// TIA Portal project "EbAndon v2_0_1" (V15)

(* hardware
DEVICE "S71500/ET200MP station_1"  S7-1500 station
   slot 0: "Rail_0"  Rack  6ES7 590-1***0-0AA0
   slot 1: "PLC_1"  CPU 1515F-2 PN  6ES7 515-2FM01-0AB0  V2.5
      slot 3: "CPU display_1"  6ES7591-1BA00-0AA0
DEVICE "HMI_1"  TP1500 Comfort PRO
   slot 0: "HMI_1"  TP1500 Comfort PRO  6AV2 124-0QC24-1AX0  15.0.0.0
   slot 1: "HMI_RT_1"  TP1500 Comfort PRO  6AV2 124-0QC24-1AX0  15.0.0.0
   slot 5: "HMI_1.IE_CP_1"  PROFINET Interface  15.0.0.0
      slot 1: "PROFINET Interface_1"  PROFINET Interface
         slot 1: "Port_1"  Port
         slot 2: "Port_2"  Port
   slot 6: "HMI_1.IE_CP_2"  PROFINET Interface  15.0.0.0
      slot 1: "PROFINET Interface_GBit"  PROFINET Interface
         slot 1: "Port_1"  Port
   slot 7: "HMI_1.MPI/DP_CP_1"  MPI/DP Interface  15.0.0.0
DEVICE "ET 200SP station_1"  ET 200SP-Station
   slot 0: "Rack_0"  Rack  6ES5 710-8MAx1
   slot 0: "volvo1606et200sp"  IM 155-6 PN ST  6ES7 155-6AU01-0BN0  V4.1
   slot 1: "DQ 8x24VDC/0.5A ST_1"  DQ 8x24VDC/0.5A ST  6ES7 132-6BF01-0BA0  V0.0
      slot 1: "DQ 8x24VDC/0.5A ST_1"  DQ 8x24VDC/0.5A ST
   slot 2: "DQ 8x24VDC/0.5A ST_2"  DQ 8x24VDC/0.5A ST  6ES7 132-6BF01-0BA0  V0.0
      slot 1: "DQ 8x24VDC/0.5A ST_2"  DQ 8x24VDC/0.5A ST
   slot 3: "DQ 8x24VDC/0.5A ST_3"  DQ 8x24VDC/0.5A ST  6ES7 132-6BF01-0BA0  V0.0
      slot 1: "DQ 8x24VDC/0.5A ST_3"  DQ 8x24VDC/0.5A ST
   slot 4: "Server module_1"  Server module  6ES7 193-6PA00-0AA0  V1.1
      slot 1: "Server module_1"  Server module
   slot 127: "BA 2xRJ45"  BA 2xRJ45  6ES7 193-6AR00-0AA0  V0.0
      slot 1: "Port_1"  6ES7 193-6AR00-0AA0  V0.0
      slot 2: "Port_2"  6ES7 193-6AR00-0AA0  V0.0
DEVICE "ET 200SP station_2"  ET 200SP-Station
   slot 0: "Rack_0"  Rack  6ES5 710-8MAx1
   slot 0: "volvo1607et200sp"  IM 155-6 PN ST  6ES7 155-6AU01-0BN0  V4.1
   slot 1: "DQ 8x24VDC/0.5A ST_1"  DQ 8x24VDC/0.5A ST  6ES7 132-6BF01-0BA0  V0.0
      slot 1: "DQ 8x24VDC/0.5A ST_1"  DQ 8x24VDC/0.5A ST
   slot 2: "DQ 8x24VDC/0.5A ST_2"  DQ 8x24VDC/0.5A ST  6ES7 132-6BF01-0BA0  V0.0
      slot 1: "DQ 8x24VDC/0.5A ST_2"  DQ 8x24VDC/0.5A ST
   slot 3: "DQ 8x24VDC/0.5A ST_3"  DQ 8x24VDC/0.5A ST  6ES7 132-6BF01-0BA0  V0.0
      slot 1: "DQ 8x24VDC/0.5A ST_3"  DQ 8x24VDC/0.5A ST
   slot 4: "Server module_1"  Server module  6ES7 193-6PA00-0AA0  V1.1
      slot 1: "Server module_1"  Server module
   slot 127: "BA 2xRJ45"  BA 2xRJ45  6ES7 193-6AR00-0AA0  V0.0
      slot 1: "Port_1"  6ES7 193-6AR00-0AA0  V0.0
      slot 2: "Port_2"  6ES7 193-6AR00-0AA0  V0.0
DEVICE "ET 200SP station_3"  ET 200SP-Station
   slot 0: "Rack_0"  Rack  6ES5 710-8MAx1
   slot 0: "volvo1608et200sp"  IM 155-6 PN ST  6ES7 155-6AU01-0BN0  V4.1
   slot 1: "DQ 8x24VDC/0.5A ST_1"  DQ 8x24VDC/0.5A ST  6ES7 132-6BF01-0BA0  V0.0
      slot 1: "DQ 8x24VDC/0.5A ST_1"  DQ 8x24VDC/0.5A ST
   slot 2: "DQ 8x24VDC/0.5A ST_2"  DQ 8x24VDC/0.5A ST  6ES7 132-6BF01-0BA0  V0.0
      slot 1: "DQ 8x24VDC/0.5A ST_2"  DQ 8x24VDC/0.5A ST
   slot 3: "DQ 8x24VDC/0.5A ST_3"  DQ 8x24VDC/0.5A ST  6ES7 132-6BF01-0BA0  V0.0
      slot 1: "DQ 8x24VDC/0.5A ST_3"  DQ 8x24VDC/0.5A ST
   slot 4: "Server module_1"  Server module  6ES7 193-6PA00-0AA0  V1.1
      slot 1: "Server module_1"  Server module
   slot 127: "BA 2xRJ45"  BA 2xRJ45  6ES7 193-6AR00-0AA0  V0.0
      slot 1: "Port_1"  6ES7 193-6AR00-0AA0  V0.0
      slot 2: "Port_2"  6ES7 193-6AR00-0AA0  V0.0
DEVICE "KP8_1"  SIMATIC Key Panel
   slot 0: "Rack"  Rail  V1.0
   slot 0: "volvo1608kp8"  KP8  6AV3 688-3AY36-0AX0  R01.00.00
DEVICE "KP8_2"  SIMATIC Key Panel
   slot 0: "Rack"  Rail  V1.0
   slot 0: "volvo1607kp8"  KP8  6AV3 688-3AY36-0AX0  R01.00.00
DEVICE "KP8_3"  SIMATIC Key Panel
   slot 0: "Rack"  Rail  V1.0
   slot 0: "volvo1606kp8"  KP8  6AV3 688-3AY36-0AX0  R01.00.00
DEVICE "KP8_4"  SIMATIC Key Panel
   slot 0: "Rack"  Rail  V1.0
   slot 0: "volvo1609kp8"  KP8  6AV3 688-3AY36-0AX0  R01.00.00
DEVICE "ET 200SP station_4"  ET 200SP-Station
   slot 0: "Rack_0"  Rack  6ES5 710-8MAx1
   slot 0: "volvo1609et200sp"  IM 155-6 PN ST  6ES7 155-6AU01-0BN0  V4.1
   slot 1: "DQ 8x24VDC/0.5A ST_1"  DQ 8x24VDC/0.5A ST  6ES7 132-6BF01-0BA0  V0.0
      slot 1: "DQ 8x24VDC/0.5A ST_1"  DQ 8x24VDC/0.5A ST
   slot 2: "DQ 8x24VDC/0.5A ST_2"  DQ 8x24VDC/0.5A ST  6ES7 132-6BF01-0BA0  V0.0
      slot 1: "DQ 8x24VDC/0.5A ST_2"  DQ 8x24VDC/0.5A ST
   slot 3: "DQ 8x24VDC/0.5A ST_3"  DQ 8x24VDC/0.5A ST  6ES7 132-6BF01-0BA0  V0.0
      slot 1: "DQ 8x24VDC/0.5A ST_3"  DQ 8x24VDC/0.5A ST
   slot 4: "Server module_1"  Server module  6ES7 193-6PA00-0AA0  V1.1
      slot 1: "Server module_1"  Server module
   slot 127: "BA 2xRJ45"  BA 2xRJ45  6ES7 193-6AR00-0AA0  V0.0
      slot 1: "Port_1"  6ES7 193-6AR00-0AA0  V0.0
      slot 2: "Port_2"  6ES7 193-6AR00-0AA0  V0.0
DEVICE "ET 200SP station_5"  ET 200SP-Station
   slot 0: "Rack_0"  Rack  6ES5 710-8MAx1
   slot 0: "volvo1610et200sp"  IM 155-6 PN ST  6ES7 155-6AU01-0BN0  V4.1
   slot 1: "DQ 8x24VDC/0.5A ST_1"  DQ 8x24VDC/0.5A ST  6ES7 132-6BF01-0BA0  V0.0
      slot 1: "DQ 8x24VDC/0.5A ST_1"  DQ 8x24VDC/0.5A ST
   slot 2: "DQ 8x24VDC/0.5A ST_2"  DQ 8x24VDC/0.5A ST  6ES7 132-6BF01-0BA0  V0.0
      slot 1: "DQ 8x24VDC/0.5A ST_2"  DQ 8x24VDC/0.5A ST
   slot 3: "DQ 8x24VDC/0.5A ST_3"  DQ 8x24VDC/0.5A ST  6ES7 132-6BF01-0BA0  V0.0
      slot 1: "DQ 8x24VDC/0.5A ST_3"  DQ 8x24VDC/0.5A ST
   slot 4: "Server module_1"  Server module  6ES7 193-6PA00-0AA0  V1.1
      slot 1: "Server module_1"  Server module
   slot 127: "BA 2xRJ45"  BA 2xRJ45  6ES7 193-6AR00-0AA0  V0.0
      slot 1: "Port_1"  6ES7 193-6AR00-0AA0  V0.0
      slot 2: "Port_2"  6ES7 193-6AR00-0AA0  V0.0
DEVICE "KP8_5"  SIMATIC Key Panel
   slot 0: "Rack"  Rail  V1.0
   slot 0: "volvo1610kp8"  KP8  6AV3 688-3AY36-0AX0  R01.00.00
DEVICE "KP8_6"  SIMATIC Key Panel
   slot 0: "Rack"  Rail  V1.0
   slot 0: "volvo1611kp8"  KP8  6AV3 688-3AY36-0AX0  R01.00.00
DEVICE "ET 200SP station_6"  ET 200SP-Station
   slot 0: "Rack_0"  Rack  6ES5 710-8MAx1
   slot 0: "volvo1611et200sp"  IM 155-6 PN ST  6ES7 155-6AU01-0BN0  V4.1
   slot 1: "DQ 8x24VDC/0.5A ST_1"  DQ 8x24VDC/0.5A ST  6ES7 132-6BF01-0BA0  V0.0
      slot 1: "DQ 8x24VDC/0.5A ST_1"  DQ 8x24VDC/0.5A ST
   slot 2: "DQ 8x24VDC/0.5A ST_2"  DQ 8x24VDC/0.5A ST  6ES7 132-6BF01-0BA0  V0.0
      slot 1: "DQ 8x24VDC/0.5A ST_2"  DQ 8x24VDC/0.5A ST
   slot 3: "DQ 8x24VDC/0.5A ST_3"  DQ 8x24VDC/0.5A ST  6ES7 132-6BF01-0BA0  V0.0
      slot 1: "DQ 8x24VDC/0.5A ST_3"  DQ 8x24VDC/0.5A ST
   slot 4: "Server module_1"  Server module  6ES7 193-6PA00-0AA0  V1.1
      slot 1: "Server module_1"  Server module
   slot 127: "BA 2xRJ45"  BA 2xRJ45  6ES7 193-6AR00-0AA0  V0.0
      slot 1: "Port_1"  6ES7 193-6AR00-0AA0  V0.0
      slot 2: "Port_2"  6ES7 193-6AR00-0AA0  V0.0
DEVICE "KP8_7"  SIMATIC Key Panel
   slot 0: "Rack"  Rail  V1.0
   slot 0: "volvo1601kp8"  KP8  6AV3 688-3AY36-0AX0  R01.00.00
DEVICE "ET 200SP station_7"  ET 200SP-Station
   slot 0: "Rack_0"  Rack  6ES5 710-8MAx1
   slot 0: "volvo1601et200sp"  IM 155-6 PN ST  6ES7 155-6AU01-0BN0  V4.1
   slot 1: "DQ 8x24VDC/0.5A ST_1"  DQ 8x24VDC/0.5A ST  6ES7 132-6BF01-0BA0  V0.0
      slot 1: "DQ 8x24VDC/0.5A ST_1"  DQ 8x24VDC/0.5A ST
   slot 2: "DQ 8x24VDC/0.5A ST_2"  DQ 8x24VDC/0.5A ST  6ES7 132-6BF01-0BA0  V0.0
      slot 1: "DQ 8x24VDC/0.5A ST_2"  DQ 8x24VDC/0.5A ST
   slot 3: "DQ 8x24VDC/0.5A ST_3"  DQ 8x24VDC/0.5A ST  6ES7 132-6BF01-0BA0  V0.0
      slot 1: "DQ 8x24VDC/0.5A ST_3"  DQ 8x24VDC/0.5A ST
   slot 4: "Server module_1"  Server module  6ES7 193-6PA00-0AA0  V1.1
      slot 1: "Server module_1"  Server module
   slot 127: "BA 2xRJ45"  BA 2xRJ45  6ES7 193-6AR00-0AA0  V0.0
      slot 1: "Port_1"  6ES7 193-6AR00-0AA0  V0.0
      slot 2: "Port_2"  6ES7 193-6AR00-0AA0  V0.0
DEVICE "ET 200SP station_8"  ET 200SP-Station
   slot 0: "Rack_0"  Rack  6ES5 710-8MAx1
   slot 0: "volvo1602et200sp"  IM 155-6 PN ST  6ES7 155-6AU01-0BN0  V4.1
   slot 1: "DQ 8x24VDC/0.5A ST_1"  DQ 8x24VDC/0.5A ST  6ES7 132-6BF01-0BA0  V0.0
      slot 1: "DQ 8x24VDC/0.5A ST_1"  DQ 8x24VDC/0.5A ST
   slot 2: "DQ 8x24VDC/0.5A ST_2"  DQ 8x24VDC/0.5A ST  6ES7 132-6BF01-0BA0  V0.0
      slot 1: "DQ 8x24VDC/0.5A ST_2"  DQ 8x24VDC/0.5A ST
   slot 3: "DQ 8x24VDC/0.5A ST_3"  DQ 8x24VDC/0.5A ST  6ES7 132-6BF01-0BA0  V0.0
      slot 1: "DQ 8x24VDC/0.5A ST_3"  DQ 8x24VDC/0.5A ST
   slot 4: "Server module_1"  Server module  6ES7 193-6PA00-0AA0  V1.1
      slot 1: "Server module_1"  Server module
   slot 127: "BA 2xRJ45"  BA 2xRJ45  6ES7 193-6AR00-0AA0  V0.0
      slot 1: "Port_1"  6ES7 193-6AR00-0AA0  V0.0
      slot 2: "Port_2"  6ES7 193-6AR00-0AA0  V0.0
DEVICE "KP8_8"  SIMATIC Key Panel
   slot 0: "Rack"  Rail  V1.0
   slot 0: "volvo1602kp8"  KP8  6AV3 688-3AY36-0AX0  R01.00.00
DEVICE "KP8_9"  SIMATIC Key Panel
   slot 0: "Rack"  Rail  V1.0
   slot 0: "volvo1603kp8"  KP8  6AV3 688-3AY36-0AX0  R01.00.00
DEVICE "KP8_10"  SIMATIC Key Panel
   slot 0: "Rack"  Rail  V1.0
   slot 0: "volvo1604kp8"  KP8  6AV3 688-3AY36-0AX0  R01.00.00
DEVICE "KP8_11"  SIMATIC Key Panel
   slot 0: "Rack"  Rail  V1.0
   slot 0: "volvo1605kp8"  KP8  6AV3 688-3AY36-0AX0  R01.00.00
DEVICE "ET 200SP station_9"  ET 200SP-Station
   slot 0: "Rack_0"  Rack  6ES5 710-8MAx1
   slot 0: "volvo1603et200sp"  IM 155-6 PN ST  6ES7 155-6AU01-0BN0  V4.1
   slot 1: "DQ 8x24VDC/0.5A ST_1"  DQ 8x24VDC/0.5A ST  6ES7 132-6BF01-0BA0  V0.0
      slot 1: "DQ 8x24VDC/0.5A ST_1"  DQ 8x24VDC/0.5A ST
   slot 2: "DQ 8x24VDC/0.5A ST_2"  DQ 8x24VDC/0.5A ST  6ES7 132-6BF01-0BA0  V0.0
      slot 1: "DQ 8x24VDC/0.5A ST_2"  DQ 8x24VDC/0.5A ST
   slot 3: "DQ 8x24VDC/0.5A ST_3"  DQ 8x24VDC/0.5A ST  6ES7 132-6BF01-0BA0  V0.0
      slot 1: "DQ 8x24VDC/0.5A ST_3"  DQ 8x24VDC/0.5A ST
   slot 4: "Server module_1"  Server module  6ES7 193-6PA00-0AA0  V1.1
      slot 1: "Server module_1"  Server module
   slot 127: "BA 2xRJ45"  BA 2xRJ45  6ES7 193-6AR00-0AA0  V0.0
      slot 1: "Port_1"  6ES7 193-6AR00-0AA0  V0.0
      slot 2: "Port_2"  6ES7 193-6AR00-0AA0  V0.0
DEVICE "ET 200SP station_10"  ET 200SP-Station
   slot 0: "Rack_0"  Rack  6ES5 710-8MAx1
   slot 0: "volvo1604et200sp"  IM 155-6 PN ST  6ES7 155-6AU01-0BN0  V4.1
   slot 1: "DQ 8x24VDC/0.5A ST_1"  DQ 8x24VDC/0.5A ST  6ES7 132-6BF01-0BA0  V0.0
      slot 1: "DQ 8x24VDC/0.5A ST_1"  DQ 8x24VDC/0.5A ST
   slot 2: "DQ 8x24VDC/0.5A ST_2"  DQ 8x24VDC/0.5A ST  6ES7 132-6BF01-0BA0  V0.0
      slot 1: "DQ 8x24VDC/0.5A ST_2"  DQ 8x24VDC/0.5A ST
   slot 3: "DQ 8x24VDC/0.5A ST_3"  DQ 8x24VDC/0.5A ST  6ES7 132-6BF01-0BA0  V0.0
      slot 1: "DQ 8x24VDC/0.5A ST_3"  DQ 8x24VDC/0.5A ST
   slot 4: "Server module_1"  Server module  6ES7 193-6PA00-0AA0  V1.1
      slot 1: "Server module_1"  Server module
   slot 127: "BA 2xRJ45"  BA 2xRJ45  6ES7 193-6AR00-0AA0  V0.0
      slot 1: "Port_1"  6ES7 193-6AR00-0AA0  V0.0
      slot 2: "Port_2"  6ES7 193-6AR00-0AA0  V0.0
DEVICE "ET 200SP station_11"  ET 200SP-Station
   slot 0: "Rack_0"  Rack  6ES5 710-8MAx1
   slot 0: "volvo1605et200sp"  IM 155-6 PN ST  6ES7 155-6AU01-0BN0  V4.1
   slot 1: "DQ 8x24VDC/0.5A ST_1"  DQ 8x24VDC/0.5A ST  6ES7 132-6BF01-0BA0  V0.0
      slot 1: "DQ 8x24VDC/0.5A ST_1"  DQ 8x24VDC/0.5A ST
   slot 2: "DQ 8x24VDC/0.5A ST_2"  DQ 8x24VDC/0.5A ST  6ES7 132-6BF01-0BA0  V0.0
      slot 1: "DQ 8x24VDC/0.5A ST_2"  DQ 8x24VDC/0.5A ST
   slot 3: "DQ 8x24VDC/0.5A ST_3"  DQ 8x24VDC/0.5A ST  6ES7 132-6BF01-0BA0  V0.0
      slot 1: "DQ 8x24VDC/0.5A ST_3"  DQ 8x24VDC/0.5A ST
   slot 4: "Server module_1"  Server module  6ES7 193-6PA00-0AA0  V1.1
      slot 1: "Server module_1"  Server module
   slot 127: "BA 2xRJ45"  BA 2xRJ45  6ES7 193-6AR00-0AA0  V0.0
      slot 1: "Port_1"  6ES7 193-6AR00-0AA0  V0.0
      slot 2: "Port_2"  6ES7 193-6AR00-0AA0  V0.0
DEVICE "PC-System_1"  SIMATIC PC station
   slot 0: "SIMATIC PC station"  Rail  SIMATIC PC-Station  V1.0
      slot 125: "Stationmanager"  Station_Manager  V6.0.4
   slot 1: "HMI_RT_2"  WinCC RT Advanced  6AV2 104-0xxxx-xxxx  15.0.0.0
      slot 33792: "Host interface"  Host interface
   slot 2: "IE general_1"  IE General  IE_CP  V8.2.0
DEVICE "ET 200SP station_12"  ET 200SP-Station
   slot 0: "Rack_0"  Rack  6ES5 710-8MAx1
   slot 0: "chm01et200sp"  IM 155-6 PN ST  6ES7 155-6AU01-0BN0  V4.1
   slot 1: "DQ 8x24VDC/0.5A ST_1"  DQ 8x24VDC/0.5A ST  6ES7 132-6BF01-0BA0  V0.0
      slot 1: "DQ 8x24VDC/0.5A ST_1"  DQ 8x24VDC/0.5A ST
   slot 2: "DQ 8x24VDC/0.5A ST_2"  DQ 8x24VDC/0.5A ST  6ES7 132-6BF01-0BA0  V0.0
      slot 1: "DQ 8x24VDC/0.5A ST_2"  DQ 8x24VDC/0.5A ST
   slot 3: "DQ 8x24VDC/0.5A ST_3"  DQ 8x24VDC/0.5A ST  6ES7 132-6BF01-0BA0  V0.0
      slot 1: "DQ 8x24VDC/0.5A ST_3"  DQ 8x24VDC/0.5A ST
   slot 4: "Server module_1"  Server module  6ES7 193-6PA00-0AA0  V1.1
      slot 1: "Server module_1"  Server module
   slot 127: "BA 2xRJ45"  BA 2xRJ45  6ES7 193-6AR00-0AA0  V0.0
      slot 1: "Port_1"  6ES7 193-6AR00-0AA0  V0.0
      slot 2: "Port_2"  6ES7 193-6AR00-0AA0  V0.0
DEVICE "KP8_12"  SIMATIC Key Panel
   slot 0: "Rack"  Rail  V1.0
   slot 0: "chm01kp8"  KP8  6AV3 688-3AY36-0AX0  R01.00.00
DEVICE "ET 200SP station_13"  ET 200SP-Station
   slot 0: "Rack_0"  Rack  6ES5 710-8MAx1
   slot 0: "chm02et200sp"  IM 155-6 PN ST  6ES7 155-6AU01-0BN0  V4.1
   slot 1: "DQ 8x24VDC/0.5A ST_1"  DQ 8x24VDC/0.5A ST  6ES7 132-6BF01-0BA0  V0.0
      slot 1: "DQ 8x24VDC/0.5A ST_1"  DQ 8x24VDC/0.5A ST
   slot 2: "DQ 8x24VDC/0.5A ST_2"  DQ 8x24VDC/0.5A ST  6ES7 132-6BF01-0BA0  V0.0
      slot 1: "DQ 8x24VDC/0.5A ST_2"  DQ 8x24VDC/0.5A ST
   slot 3: "DQ 8x24VDC/0.5A ST_3"  DQ 8x24VDC/0.5A ST  6ES7 132-6BF01-0BA0  V0.0
      slot 1: "DQ 8x24VDC/0.5A ST_3"  DQ 8x24VDC/0.5A ST
   slot 4: "Server module_1"  Server module  6ES7 193-6PA00-0AA0  V1.1
      slot 1: "Server module_1"  Server module
   slot 127: "BA 2xRJ45"  BA 2xRJ45  6ES7 193-6AR00-0AA0  V0.0
      slot 1: "Port_1"  6ES7 193-6AR00-0AA0  V0.0
      slot 2: "Port_2"  6ES7 193-6AR00-0AA0  V0.0
DEVICE "KP8_13"  SIMATIC Key Panel
   slot 0: "Rack"  Rail  V1.0
   slot 0: "chm02kp8"  KP8  6AV3 688-3AY36-0AX0  R01.00.00
DEVICE "ET 200SP station_14"  ET 200SP-Station
   slot 0: "Rack_0"  Rack  6ES5 710-8MAx1
   slot 0: "chm03et200sp"  IM 155-6 PN ST  6ES7 155-6AU01-0BN0  V4.1
   slot 1: "DQ 8x24VDC/0.5A ST_1"  DQ 8x24VDC/0.5A ST  6ES7 132-6BF01-0BA0  V0.0
      slot 1: "DQ 8x24VDC/0.5A ST_1"  DQ 8x24VDC/0.5A ST
   slot 2: "DQ 8x24VDC/0.5A ST_2"  DQ 8x24VDC/0.5A ST  6ES7 132-6BF01-0BA0  V0.0
      slot 1: "DQ 8x24VDC/0.5A ST_2"  DQ 8x24VDC/0.5A ST
   slot 3: "DQ 8x24VDC/0.5A ST_3"  DQ 8x24VDC/0.5A ST  6ES7 132-6BF01-0BA0  V0.0
      slot 1: "DQ 8x24VDC/0.5A ST_3"  DQ 8x24VDC/0.5A ST
   slot 4: "Server module_1"  Server module  6ES7 193-6PA00-0AA0  V1.1
      slot 1: "Server module_1"  Server module
   slot 127: "BA 2xRJ45"  BA 2xRJ45  6ES7 193-6AR00-0AA0  V0.0
      slot 1: "Port_1"  6ES7 193-6AR00-0AA0  V0.0
      slot 2: "Port_2"  6ES7 193-6AR00-0AA0  V0.0
DEVICE "KP8_14"  SIMATIC Key Panel
   slot 0: "Rack"  Rail  V1.0
   slot 0: "chm03kp8"  KP8  6AV3 688-3AY36-0AX0  R01.00.00
DEVICE "KP8_15"  SIMATIC Key Panel
   slot 0: "Rack"  Rail  V1.0
   slot 0: "chm04kp8"  KP8  6AV3 688-3AY36-0AX0  R01.00.00
DEVICE "ET 200SP station_15"  ET 200SP-Station
   slot 0: "Rack_0"  Rack  6ES5 710-8MAx1
   slot 0: "chm04et200sp"  IM 155-6 PN ST  6ES7 155-6AU01-0BN0  V4.1
   slot 1: "DQ 8x24VDC/0.5A ST_1"  DQ 8x24VDC/0.5A ST  6ES7 132-6BF01-0BA0  V0.0
      slot 1: "DQ 8x24VDC/0.5A ST_1"  DQ 8x24VDC/0.5A ST
   slot 2: "DQ 8x24VDC/0.5A ST_2"  DQ 8x24VDC/0.5A ST  6ES7 132-6BF01-0BA0  V0.0
      slot 1: "DQ 8x24VDC/0.5A ST_2"  DQ 8x24VDC/0.5A ST
   slot 3: "DQ 8x24VDC/0.5A ST_3"  DQ 8x24VDC/0.5A ST  6ES7 132-6BF01-0BA0  V0.0
      slot 1: "DQ 8x24VDC/0.5A ST_3"  DQ 8x24VDC/0.5A ST
   slot 4: "Server module_1"  Server module  6ES7 193-6PA00-0AA0  V1.1
      slot 1: "Server module_1"  Server module
   slot 127: "BA 2xRJ45"  BA 2xRJ45  6ES7 193-6AR00-0AA0  V0.0
      slot 1: "Port_1"  6ES7 193-6AR00-0AA0  V0.0
      slot 2: "Port_2"  6ES7 193-6AR00-0AA0  V0.0
DEVICE "KP8_16"  SIMATIC Key Panel
   slot 0: "Rack"  Rail  V1.0
   slot 0: "cdo01kp8"  KP8  6AV3 688-3AY36-0AX0  R01.00.00
DEVICE "ET 200SP station_16"  ET 200SP-Station
   slot 0: "Rack_0"  Rack  6ES5 710-8MAx1
   slot 0: "cdo01et200sp"  IM 155-6 PN ST  6ES7 155-6AU01-0BN0  V4.1
   slot 1: "DQ 8x24VDC/0.5A ST_1"  DQ 8x24VDC/0.5A ST  6ES7 132-6BF01-0BA0  V0.0
      slot 1: "DQ 8x24VDC/0.5A ST_1"  DQ 8x24VDC/0.5A ST
   slot 2: "DQ 8x24VDC/0.5A ST_2"  DQ 8x24VDC/0.5A ST  6ES7 132-6BF01-0BA0  V0.0
      slot 1: "DQ 8x24VDC/0.5A ST_2"  DQ 8x24VDC/0.5A ST
   slot 3: "DQ 8x24VDC/0.5A ST_3"  DQ 8x24VDC/0.5A ST  6ES7 132-6BF01-0BA0  V0.0
      slot 1: "DQ 8x24VDC/0.5A ST_3"  DQ 8x24VDC/0.5A ST
   slot 4: "Server module_1"  Server module  6ES7 193-6PA00-0AA0  V1.1
      slot 1: "Server module_1"  Server module
   slot 127: "BA 2xRJ45"  BA 2xRJ45  6ES7 193-6AR00-0AA0  V0.0
      slot 1: "Port_1"  6ES7 193-6AR00-0AA0  V0.0
      slot 2: "Port_2"  6ES7 193-6AR00-0AA0  V0.0
DEVICE "ET 200SP station_17"  ET 200SP-Station
   slot 0: "Rack_0"  Rack  6ES5 710-8MAx1
   slot 0: "cdo02et200sp"  IM 155-6 PN ST  6ES7 155-6AU01-0BN0  V4.1
   slot 1: "DQ 8x24VDC/0.5A ST_1"  DQ 8x24VDC/0.5A ST  6ES7 132-6BF01-0BA0  V0.0
      slot 1: "DQ 8x24VDC/0.5A ST_1"  DQ 8x24VDC/0.5A ST
   slot 2: "DQ 8x24VDC/0.5A ST_2"  DQ 8x24VDC/0.5A ST  6ES7 132-6BF01-0BA0  V0.0
      slot 1: "DQ 8x24VDC/0.5A ST_2"  DQ 8x24VDC/0.5A ST
   slot 3: "DQ 8x24VDC/0.5A ST_3"  DQ 8x24VDC/0.5A ST  6ES7 132-6BF01-0BA0  V0.0
      slot 1: "DQ 8x24VDC/0.5A ST_3"  DQ 8x24VDC/0.5A ST
   slot 4: "Server module_1"  Server module  6ES7 193-6PA00-0AA0  V1.1
      slot 1: "Server module_1"  Server module
   slot 127: "BA 2xRJ45"  BA 2xRJ45  6ES7 193-6AR00-0AA0  V0.0
      slot 1: "Port_1"  6ES7 193-6AR00-0AA0  V0.0
      slot 2: "Port_2"  6ES7 193-6AR00-0AA0  V0.0
DEVICE "KP8_17"  SIMATIC Key Panel
   slot 0: "Rack"  Rail  V1.0
   slot 0: "cdo02kp8"  KP8  6AV3 688-3AY36-0AX0  R01.00.00
DEVICE "KP8_18"  SIMATIC Key Panel
   slot 0: "Rack"  Rail  V1.0
   slot 0: "cdo03kp8"  KP8  6AV3 688-3AY36-0AX0  R01.00.00
DEVICE "ET 200SP station_18"  ET 200SP-Station
   slot 0: "Rack_0"  Rack  6ES5 710-8MAx1
   slot 0: "cdo03et200sp"  IM 155-6 PN ST  6ES7 155-6AU01-0BN0  V4.1
   slot 1: "DQ 8x24VDC/0.5A ST_1"  DQ 8x24VDC/0.5A ST  6ES7 132-6BF01-0BA0  V0.0
      slot 1: "DQ 8x24VDC/0.5A ST_1"  DQ 8x24VDC/0.5A ST
   slot 2: "DQ 8x24VDC/0.5A ST_2"  DQ 8x24VDC/0.5A ST  6ES7 132-6BF01-0BA0  V0.0
      slot 1: "DQ 8x24VDC/0.5A ST_2"  DQ 8x24VDC/0.5A ST
   slot 3: "DQ 8x24VDC/0.5A ST_3"  DQ 8x24VDC/0.5A ST  6ES7 132-6BF01-0BA0  V0.0
      slot 1: "DQ 8x24VDC/0.5A ST_3"  DQ 8x24VDC/0.5A ST
   slot 4: "Server module_1"  Server module  6ES7 193-6PA00-0AA0  V1.1
      slot 1: "Server module_1"  Server module
   slot 127: "BA 2xRJ45"  BA 2xRJ45  6ES7 193-6AR00-0AA0  V0.0
      slot 1: "Port_1"  6ES7 193-6AR00-0AA0  V0.0
      slot 2: "Port_2"  6ES7 193-6AR00-0AA0  V0.0
DEVICE "ET 200SP station_19"  ET 200SP-Station
   slot 0: "Rack_0"  Rack  6ES5 710-8MAx1
   slot 0: "bfl01et200sp"  IM 155-6 PN ST  6ES7 155-6AU01-0BN0  V4.1
   slot 1: "DQ 8x24VDC/0.5A ST_1"  DQ 8x24VDC/0.5A ST  6ES7 132-6BF01-0BA0  V0.0
      slot 1: "DQ 8x24VDC/0.5A ST_1"  DQ 8x24VDC/0.5A ST
   slot 2: "DQ 8x24VDC/0.5A ST_2"  DQ 8x24VDC/0.5A ST  6ES7 132-6BF01-0BA0  V0.0
      slot 1: "DQ 8x24VDC/0.5A ST_2"  DQ 8x24VDC/0.5A ST
   slot 3: "DQ 8x24VDC/0.5A ST_3"  DQ 8x24VDC/0.5A ST  6ES7 132-6BF01-0BA0  V0.0
      slot 1: "DQ 8x24VDC/0.5A ST_3"  DQ 8x24VDC/0.5A ST
   slot 4: "Server module_1"  Server module  6ES7 193-6PA00-0AA0  V1.1
      slot 1: "Server module_1"  Server module
   slot 127: "BA 2xRJ45"  BA 2xRJ45  6ES7 193-6AR00-0AA0  V0.0
      slot 1: "Port_1"  6ES7 193-6AR00-0AA0  V0.0
      slot 2: "Port_2"  6ES7 193-6AR00-0AA0  V0.0
DEVICE "KP8_19"  SIMATIC Key Panel
   slot 0: "Rack"  Rail  V1.0
   slot 0: "bfl01kp8"  KP8  6AV3 688-3AY36-0AX0  R01.00.00
DEVICE "KP8_20"  SIMATIC Key Panel
   slot 0: "Rack"  Rail  V1.0
   slot 0: "bfl02kp8"  KP8  6AV3 688-3AY36-0AX0  R01.00.00
DEVICE "ET 200SP station_20"  ET 200SP-Station
   slot 0: "Rack_0"  Rack  6ES5 710-8MAx1
   slot 0: "bfl02et200sp"  IM 155-6 PN ST  6ES7 155-6AU01-0BN0  V4.1
   slot 1: "DQ 8x24VDC/0.5A ST_1"  DQ 8x24VDC/0.5A ST  6ES7 132-6BF01-0BA0  V0.0
      slot 1: "DQ 8x24VDC/0.5A ST_1"  DQ 8x24VDC/0.5A ST
   slot 2: "DQ 8x24VDC/0.5A ST_2"  DQ 8x24VDC/0.5A ST  6ES7 132-6BF01-0BA0  V0.0
      slot 1: "DQ 8x24VDC/0.5A ST_2"  DQ 8x24VDC/0.5A ST
   slot 3: "DQ 8x24VDC/0.5A ST_3"  DQ 8x24VDC/0.5A ST  6ES7 132-6BF01-0BA0  V0.0
      slot 1: "DQ 8x24VDC/0.5A ST_3"  DQ 8x24VDC/0.5A ST
   slot 4: "Server module_1"  Server module  6ES7 193-6PA00-0AA0  V1.1
      slot 1: "Server module_1"  Server module
   slot 127: "BA 2xRJ45"  BA 2xRJ45  6ES7 193-6AR00-0AA0  V0.0
      slot 1: "Port_1"  6ES7 193-6AR00-0AA0  V0.0
      slot 2: "Port_2"  6ES7 193-6AR00-0AA0  V0.0
DEVICE "ET 200SP station_21"  ET 200SP-Station
   slot 0: "Rack_0"  Rack  6ES5 710-8MAx1
   slot 0: "bfl03et200sp"  IM 155-6 PN ST  6ES7 155-6AU01-0BN0  V4.1
   slot 1: "DQ 8x24VDC/0.5A ST_1"  DQ 8x24VDC/0.5A ST  6ES7 132-6BF01-0BA0  V0.0
      slot 1: "DQ 8x24VDC/0.5A ST_1"  DQ 8x24VDC/0.5A ST
   slot 2: "DQ 8x24VDC/0.5A ST_2"  DQ 8x24VDC/0.5A ST  6ES7 132-6BF01-0BA0  V0.0
      slot 1: "DQ 8x24VDC/0.5A ST_2"  DQ 8x24VDC/0.5A ST
   slot 3: "DQ 8x24VDC/0.5A ST_3"  DQ 8x24VDC/0.5A ST  6ES7 132-6BF01-0BA0  V0.0
      slot 1: "DQ 8x24VDC/0.5A ST_3"  DQ 8x24VDC/0.5A ST
   slot 4: "Server module_1"  Server module  6ES7 193-6PA00-0AA0  V1.1
      slot 1: "Server module_1"  Server module
   slot 127: "BA 2xRJ45"  BA 2xRJ45  6ES7 193-6AR00-0AA0  V0.0
      slot 1: "Port_1"  6ES7 193-6AR00-0AA0  V0.0
      slot 2: "Port_2"  6ES7 193-6AR00-0AA0  V0.0
DEVICE "KP8_21"  SIMATIC Key Panel
   slot 0: "Rack"  Rail  V1.0
   slot 0: "bfl03kp8"  KP8  6AV3 688-3AY36-0AX0  R01.00.00
DEVICE "KP8_22"  SIMATIC Key Panel
   slot 0: "Rack"  Rail  V1.0
   slot 0: "lgs01kp8"  KP8  6AV3 688-3AY36-0AX0  R01.00.00
DEVICE "ET 200SP station_22"  ET 200SP-Station
   slot 0: "Rack_0"  Rack  6ES5 710-8MAx1
   slot 0: "lgs01et200sp"  IM 155-6 PN ST  6ES7 155-6AU01-0BN0  V4.1
   slot 1: "DQ 8x24VDC/0.5A ST_1"  DQ 8x24VDC/0.5A ST  6ES7 132-6BF01-0BA0  V0.0
      slot 1: "DQ 8x24VDC/0.5A ST_1"  DQ 8x24VDC/0.5A ST
   slot 2: "DQ 8x24VDC/0.5A ST_2"  DQ 8x24VDC/0.5A ST  6ES7 132-6BF01-0BA0  V0.0
      slot 1: "DQ 8x24VDC/0.5A ST_2"  DQ 8x24VDC/0.5A ST
   slot 3: "DQ 8x24VDC/0.5A ST_3"  DQ 8x24VDC/0.5A ST  6ES7 132-6BF01-0BA0  V0.0
      slot 1: "DQ 8x24VDC/0.5A ST_3"  DQ 8x24VDC/0.5A ST
   slot 4: "Server module_1"  Server module  6ES7 193-6PA00-0AA0  V1.1
      slot 1: "Server module_1"  Server module
   slot 127: "BA 2xRJ45"  BA 2xRJ45  6ES7 193-6AR00-0AA0  V0.0
      slot 1: "Port_1"  6ES7 193-6AR00-0AA0  V0.0
      slot 2: "Port_2"  6ES7 193-6AR00-0AA0  V0.0
DEVICE "ET 200SP station_23"  ET 200SP-Station
   slot 0: "Rack_0"  Rack  6ES5 710-8MAx1
   slot 0: "lgs02et200sp"  IM 155-6 PN ST  6ES7 155-6AU01-0BN0  V4.1
   slot 1: "DQ 8x24VDC/0.5A ST_1"  DQ 8x24VDC/0.5A ST  6ES7 132-6BF01-0BA0  V0.0
      slot 1: "DQ 8x24VDC/0.5A ST_1"  DQ 8x24VDC/0.5A ST
   slot 2: "DQ 8x24VDC/0.5A ST_2"  DQ 8x24VDC/0.5A ST  6ES7 132-6BF01-0BA0  V0.0
      slot 1: "DQ 8x24VDC/0.5A ST_2"  DQ 8x24VDC/0.5A ST
   slot 3: "DQ 8x24VDC/0.5A ST_3"  DQ 8x24VDC/0.5A ST  6ES7 132-6BF01-0BA0  V0.0
      slot 1: "DQ 8x24VDC/0.5A ST_3"  DQ 8x24VDC/0.5A ST
   slot 4: "Server module_1"  Server module  6ES7 193-6PA00-0AA0  V1.1
      slot 1: "Server module_1"  Server module
   slot 127: "BA 2xRJ45"  BA 2xRJ45  6ES7 193-6AR00-0AA0  V0.0
      slot 1: "Port_1"  6ES7 193-6AR00-0AA0  V0.0
      slot 2: "Port_2"  6ES7 193-6AR00-0AA0  V0.0
DEVICE "KP8_23"  SIMATIC Key Panel
   slot 0: "Rack"  Rail  V1.0
   slot 0: "lgs02kp8"  KP8  6AV3 688-3AY36-0AX0  R01.00.00
DEVICE "KP8_24"  SIMATIC Key Panel
   slot 0: "Rack"  Rail  V1.0
   slot 0: "chm05kp8"  KP8  6AV3 688-3AY36-0AX0  R01.00.00
DEVICE "ET 200SP station_24"  ET 200SP-Station
   slot 0: "Rack_0"  Rack  6ES5 710-8MAx1
   slot 0: "chm05et200sp"  IM 155-6 PN ST  6ES7 155-6AU01-0BN0  V4.1
   slot 1: "DQ 8x24VDC/0.5A ST_1"  DQ 8x24VDC/0.5A ST  6ES7 132-6BF01-0BA0  V0.0
      slot 1: "DQ 8x24VDC/0.5A ST_1"  DQ 8x24VDC/0.5A ST
   slot 2: "DQ 8x24VDC/0.5A ST_2"  DQ 8x24VDC/0.5A ST  6ES7 132-6BF01-0BA0  V0.0
      slot 1: "DQ 8x24VDC/0.5A ST_2"  DQ 8x24VDC/0.5A ST
   slot 3: "DQ 8x24VDC/0.5A ST_3"  DQ 8x24VDC/0.5A ST  6ES7 132-6BF01-0BA0  V0.0
      slot 1: "DQ 8x24VDC/0.5A ST_3"  DQ 8x24VDC/0.5A ST
   slot 4: "Server module_1"  Server module  6ES7 193-6PA00-0AA0  V1.1
      slot 1: "Server module_1"  Server module
   slot 127: "BA 2xRJ45"  BA 2xRJ45  6ES7 193-6AR00-0AA0  V0.0
      slot 1: "Port_1"  6ES7 193-6AR00-0AA0  V0.0
      slot 2: "Port_2"  6ES7 193-6AR00-0AA0  V0.0
*)

// ===== PLC "PLC_1"  CPU 1515F-2 PN =====

VAR_GLOBAL   // PLC tag table "Default tag table"
   "System_Byte" AT %MB1 : Byte;
   "FirstScan" AT %M1.0 : Bool;
   "DiagStatusUpdate" AT %M1.1 : Bool;
   "AlwaysTRUE" AT %M1.2 : Bool;
   "AlwaysFALSE" AT %M1.3 : Bool;
   "Clock_Byte" AT %MB0 : Byte;
   "Clock_10Hz" AT %M0.0 : Bool;
   "Clock_5Hz" AT %M0.1 : Bool;
   "Clock_2.5Hz" AT %M0.2 : Bool;
   "Clock_2Hz" AT %M0.3 : Bool;
   "Clock_1.25Hz" AT %M0.4 : Bool;
   "Clock_1Hz" AT %M0.5 : Bool;
   "Clock_0.625Hz" AT %M0.6 : Bool;
   "Clock_0.5Hz" AT %M0.7 : Bool;
   "Temp Reset" AT %M2.0 : Bool;
   "clearPartData" AT %M100.0 : Bool;
   "setDefaultPresets" AT %M100.1 : Bool;
   "hardInitReq" AT %M100.2 : Bool;
END_VAR

VAR_GLOBAL   // PLC tag table "VOLVO 16 01"
   "VOLVO 16 01 IO" AT %QD100 : DWord;
   "VOLVO 16 01 KP8 In" AT %ID0 : DWord;
   "VOLVO 16 01 KP8 Out" AT %QD0 : DWord;
END_VAR

VAR_GLOBAL   // PLC tag table "VOLVO 16 02"
   "VOLVO 16 02 IO" AT %QD104 : DWord;
   "VOLVO 16 02 KP8 In" AT %ID4 : DWord;
   "VOLVO 16 02 KP8 Out" AT %QD4 : DWord;
END_VAR

VAR_GLOBAL   // PLC tag table "VOLVO 16 03"
   "VOLVO 16 03 IO" AT %QD108 : DWord;
   "VOLVO 16 03 KP8 In" AT %ID8 : DWord;
   "VOLVO 16 03 KP8 Out" AT %QD8 : DWord;
END_VAR

VAR_GLOBAL   // PLC tag table "VOLVO 16 04"
   "VOLVO 16 04 IO" AT %QD112 : DWord;
   "VOLVO 16 04 KP8 In" AT %ID12 : DWord;
   "VOLVO 16 04 KP8 Out" AT %QD12 : DWord;
END_VAR

VAR_GLOBAL   // PLC tag table "VOLVO 16 05"
   "VOLVO 16 05 IO" AT %QD116 : DWord;
   "VOLVO 16 05 KP8 In" AT %ID16 : DWord;
   "VOLVO 16 05 KP8 Out" AT %QD16 : DWord;
END_VAR

VAR_GLOBAL   // PLC tag table "VOLVO 16 06"
   "VOLVO 16 06 IO" AT %QD120 : DWord;
   "VOLVO 16 06 KP8 In" AT %ID20 : DWord;
   "VOLVO 16 06 KP8 Out" AT %QD20 : DWord;
END_VAR

VAR_GLOBAL   // PLC tag table "VOLVO 16 07"
   "VOLVO 16 07 IO" AT %QD124 : DWord;
   "VOLVO 16 07 KP8 In" AT %ID24 : DWord;
   "VOLVO 16 07 KP8 Out" AT %QD24 : DWord;
END_VAR

VAR_GLOBAL   // PLC tag table "VOLVO 16 08"
   "VOLVO 16 08 IO" AT %QD128 : DWord;
   "VOLVO 16 08 KP8 In" AT %ID28 : DWord;
   "VOLVO 16 08 KP8 Out" AT %QD28 : DWord;
END_VAR

VAR_GLOBAL   // PLC tag table "VOLVO 16 09"
   "VOLVO 16 09 IO" AT %QD132 : DWord;
   "VOLVO 16 09 KP8 In" AT %ID32 : DWord;
   "VOLVO 16 09 KP8 Out" AT %QD32 : DWord;
END_VAR

VAR_GLOBAL   // PLC tag table "VOLVO 16 10"
   "VOLVO 16 10 IO" AT %QD136 : DWord;
   "VOLVO 16 10 KP8 In" AT %ID36 : DWord;
   "VOLVO 16 10 KP8 Out" AT %QD36 : DWord;
END_VAR

VAR_GLOBAL   // PLC tag table "VOLVO 16 11"
   "VOLVO 16 11 IO" AT %QD140 : DWord;
   "VOLVO 16 11 KP8 In" AT %ID40 : DWord;
   "VOLVO 16 11 KP8 Out" AT %QD40 : DWord;
END_VAR

VAR_GLOBAL   // PLC tag table "CHM 02"
   "CHM 02 KP8 In" AT %ID44 : DWord;
   "CHM 02 KP8 Out" AT %QD44 : DWord;
   "CHM 02 IO" AT %QD144 : DWord;
END_VAR

VAR_GLOBAL   // PLC tag table "CHM 03"
   "CHM 03 IO" AT %QD148 : DWord;
   "CHM 03 KP8 In" AT %ID48 : DWord;
   "CHM 03 KP8 Out" AT %QD48 : DWord;
END_VAR

VAR_GLOBAL   // PLC tag table "CHM 04"
   "CHM 04 IO" AT %QD152 : DWord;
   "CHM 04 KP8 In" AT %ID52 : DWord;
   "CHM 04 KP8 Out" AT %QD52 : DWord;
END_VAR

VAR_GLOBAL   // PLC tag table "CHM 05"
   "CHM 05 IO" AT %QD156 : DWord;
   "CHM 05 KP8 In" AT %ID56 : DWord;
   "CHM 05 KP8 Out" AT %QD56 : DWord;
END_VAR

VAR_GLOBAL   // PLC tag table "CDO 01"
   "CDO 01 IO" AT %QD160 : DWord;
   "CDO 01 KP8 In" AT %ID60 : DWord;
   "CDO 01 KP8 Out" AT %QD60 : DWord;
END_VAR

VAR_GLOBAL   // PLC tag table "CDO 02"
   "CDO 02 IO" AT %QD164 : DWord;
   "CDO 02 KP8 In" AT %ID64 : DWord;
   "CDO 02 KP8 Out" AT %QD64 : DWord;
END_VAR

VAR_GLOBAL   // PLC tag table "CDO 03"
   "CDO 03 IO" AT %QD168 : DWord;
   "CDO 03 KP8 In" AT %ID68 : DWord;
   "CDO 03 KP8 Out" AT %QD68 : DWord;
END_VAR

VAR_GLOBAL   // PLC tag table "BFL 01"
   "BFL 01 IO" AT %QD172 : DWord;
   "BFL 01 KP8 In" AT %ID72 : DWord;
   "BFL 01 KP8 Out" AT %QD72 : DWord;
END_VAR

VAR_GLOBAL   // PLC tag table "BFL 02"
   "BFL 02 IO" AT %QD176 : DWord;
   "BFL 02 KP8 In" AT %ID76 : DWord;
   "BFL 02 KP8 Out" AT %QD76 : DWord;
END_VAR

VAR_GLOBAL   // PLC tag table "BFL 03"
   "BFL 03 IO" AT %QD180 : DWord;
   "BFL 03 KP8 In" AT %ID80 : DWord;
   "BFL 03 KP8 Out" AT %QD80 : DWord;
END_VAR

VAR_GLOBAL   // PLC tag table "LGS 01"
   "LGS 01 IO" AT %QD184 : DWord;
   "LGS 01 KP8 In" AT %ID84 : DWord;
   "LGS 01 KP8 Out" AT %QD84 : DWord;
END_VAR

VAR_GLOBAL   // PLC tag table "LGS 02"
   "LGS 02 IO" AT %QD188 : DWord;
   "LGS 02 KP8 In" AT %ID88 : DWord;
   "LGS 02 KP8 Out" AT %QD88 : DWord;
END_VAR

VAR_GLOBAL   // PLC tag table "CHM 01"
   "CHM 01 IO" AT %QD192 : DWord;
   "CHM 01 KP8 In" AT %ID92 : DWord;
   "CHM 01 KP8 Out" AT %QD92 : DWord;
END_VAR

TYPE "Stations"
   STRUCT
      current : Array[0..23] of "Station";
      old : Array[0..23] of "Station";
   END_STRUCT;
END_TYPE

TYPE "Part Call Screen"
   STRUCT
      current : Array[0..11] of "Table Row";
   END_STRUCT;
END_TYPE

TYPE "Settings Screen"
   STRUCT
      current : "Settings";
   END_STRUCT;
END_TYPE

TYPE "Barcode Screen"
   STRUCT
      partNumber : WString[40];
      barcode : String;
      orderCancelled : Bool;
      ordered : Bool;
   END_STRUCT;
END_TYPE

TYPE "Table Row"
   STRUCT
      address : UInt;
      ordered : Bool;
      pbSelection : Struct
         actuate : Bool;
         animate : USInt;
      END_STRUCT;
      rtBackground : Struct
         animate : USInt;
      END_STRUCT;
      tfDropZone : Struct
         animate : USInt;
         value : WString[20];
      END_STRUCT;
      tfLine : Struct
         animate : USInt;
         value : WString[20];
      END_STRUCT;
      tfPartNumber : Struct
         animate : USInt;
         value : WString[40];
      END_STRUCT;
      tfTime : Struct
         animate : UInt;
         value : WString[20];
      END_STRUCT;
   END_STRUCT;
END_TYPE

TYPE "Runtime Data"
   STRUCT
      asReal : Real;
      elapsed : LReal;
      mem : LReal;
   END_STRUCT;
END_TYPE

TYPE "KP8 Button Config"
   STRUCT
      activate : Array[0..7] of Bool;
      colorOn1 : Array[0..7] of String[10];
      colorOn2 : Array[0..7] of String[10];
      colorOff : Array[0..7] of String[10];
      flash : Array[0..7] of Bool;
      group : Array[0..7] of Int;
      mode : Array[0..7] of Bool;
   END_STRUCT;
END_TYPE

TYPE "Constants"
   STRUCT
      buttonCount : Int := 6;   // max buttons per station
      hmiRowCount : Int := 11;   // number of rows displayed on hmi
      stationCount : Int := 24;   // total number of stations
      hmiSelStnCount : Int := 12;   // labels for settings screen
      defaultAlotted : Real := 1800.0;
      defaultCritical : Real := 300.0;
      partReqRows : Int := 200;
      ledRowCount : Int := 11;
      colorLib : "Color Library";
   END_STRUCT;
END_TYPE

TYPE "Part Request Data"
   STRUCT
      row : Array[0..199] of "Table Row";
   END_STRUCT;
END_TYPE

TYPE "Station"
   STRUCT
      animations : Array[0..7] of Int;
      btnStates : Array[0..7] of Bool;
      dropZone : USInt;
      elapsedTime : Struct
         partReq : Array[0..7] of Real;
         resetReq : Real;
      END_STRUCT;
      kp8Config : "KP8 Button Config";
      kp8In : Byte;
      kp8Out : DWord;
      init : Struct
         hard : Bool;
         soft : Bool;
      END_STRUCT;
      line : WString[20];
      partNumbers : Array[0..7] of WString[40];
      partOrdered : Array[0..7] of Bool;
      presetTime : Struct
         allotted : Array[0..7] of Real;
         critical : Array[0..7] of Real;
      END_STRUCT;
      stackLightOut : DWord;
      settings : Struct
         selected : Bool;
         btnSelection : Array[0..7] of Bool;
      END_STRUCT;
   END_STRUCT;
END_TYPE

TYPE "Settings"
   STRUCT
      alotted : Struct
         assign : "PB Data: Text Label";
         ioField : "IO Field Data: Timers";
      END_STRUCT;
      critical : Struct
         assign : "PB Data: Text Label";
         ioField : "IO Field Data: Timers";
      END_STRUCT;
      kp8 : Struct
         selectButtons : "PB Data: Text Label";
         btnSelState : Array[0..7] of Bool;
         buttons : Array[0..7] of "PB Data: Text Label";
         selBtnNumber : Int;
         selCount : Int;
      END_STRUCT;
      stations : Struct
         selectAll : "PB Data: Text Label";
         nextGroup : "PB Data: Graphic/Text List";
         prevGroup : "PB Data: Graphic/Text List";
         selectBtns : Array[0..11] of "PB Data: Text Label";
         selCount : Int;
      END_STRUCT;
      partNumber : Struct
         assign : "PB Data: Text Label";
         ioField : "IO Field Data: Part Number";
      END_STRUCT;
      viewingStation : Struct
         btns : Array[0..5] of "Station Assignment: Button Details";
         dzData : "Drop Zone Data";
         lineData : "Line Label Data";
         next : "PB Data: Graphic/Text List";
         previous : "PB Data: Graphic/Text List";
         "name" : WString[20];
      END_STRUCT;
   END_STRUCT;
END_TYPE

TYPE "PB Data: Graphic/Text List"
   STRUCT
      actuate : Bool;
      animate : USInt;
      listSelect : UInt;
   END_STRUCT;
END_TYPE

TYPE "LED Sign Data"
   STRUCT
      row : Array[0..11] of "Table Row";
   END_STRUCT;
END_TYPE

TYPE "PB Data: Text Label"
   STRUCT
      actuate : Bool;
      animate : USInt;
      label : WString[20];
   END_STRUCT;
END_TYPE

TYPE "Color Library"
   STRUCT
      BkBk : USInt := 0;
      BgWh : USInt := 1;
      FgWh : USInt := 2;
      FlWh : USInt := 3;
      BgGray : USInt := 4;
      FgGray : USInt := 5;
      FlGray : USInt := 6;
      BgLRd : USInt := 7;
      FgLRd : USInt := 8;
      FlLRd : USInt := 9;
      BgDRd : USInt := 10;
      FgDRd : USInt := 11;
      FlDrd : USInt := 12;
      BgLYe : USInt := 13;
      FgLYe : USInt := 14;
      FlLYe : USInt := 15;
      BgDYe : USInt := 16;
      FgDYe : USInt := 17;
      FlDYe : USInt := 18;
      BgLGr : USInt := 19;
      FgLGr : USInt := 20;
      FlLGr : USInt := 21;
      BgDGr : USInt := 22;
      FgDGr : USInt := 23;
      FlDGr : USInt := 24;
      BgLTe : USInt := 25;
      FgLTe : USInt := 26;
      FlLTe : USInt := 27;
      BgDTe : USInt := 28;
      FgDTe : USInt := 29;
      FlDTe : USInt := 30;
      BgLBl : USInt := 31;
      FgLBl : USInt := 32;
      FlLBl : USInt := 33;
      BgDBl : USInt := 34;
      FgDBl : USInt := 35;
      FlDBl : USInt := 36;
      BgLPu : USInt := 37;
      FgLPu : USInt := 38;
      FlLPu : USInt := 39;
      BgDPu : USInt := 40;
      FgDPu : USInt := 41;
      FlDPu : USInt := 42;
      disabled : USInt := 254;
      invisible : USInt := 255;
   END_STRUCT;
END_TYPE

TYPE "Station Assignment: Button Details"
   STRUCT
      alloted : Struct
         animate : USInt;
         value : WString[10];
      END_STRUCT;
      critical : Struct
         animate : USInt;
         value : WString[10];
      END_STRUCT;
      label : Struct
         animate : USInt;
         value : WString[2];
      END_STRUCT;
      partNumber : Struct
         animate : USInt;
         value : WString[40];
      END_STRUCT;
      select : Struct
         actuate : Bool;
         animate : USInt;
      END_STRUCT;
   END_STRUCT;
END_TYPE

TYPE "IO Field Data: Part Number"
   STRUCT
      animate : USInt;
      inputFinished : Bool;
      value : WString[40];
   END_STRUCT;
END_TYPE

TYPE "Line Label Data"
   STRUCT
      animate : Struct
         bg : USInt;
         ioField : USInt;
      END_STRUCT;
      inputFinished : Bool;
      value : WString[10];
   END_STRUCT;
END_TYPE

TYPE "Drop Zone Data"
   STRUCT
      animate : Struct
         bg : USInt;
         ioField : USInt;
      END_STRUCT;
      inputFinished : Bool;
      value : WString[10];
   END_STRUCT;
END_TYPE

TYPE "IO Field Data: Timers"
   STRUCT
      animate : USInt;
      inputFinished : Bool;
      value : WString[5];
   END_STRUCT;
END_TYPE

DATA_BLOCK "EMP IDB"   // DB1
{ S7_Optimized_Access := 'TRUE' }
VERSION : 0.1
// stored: InstanceOfName EMP
"EMP"
BEGIN
   constants.buttonCount := 8;
   stations.current[0].presetTime.allotted[7] := 1800.0;
   stations.current[0].presetTime.allotted[3] := 1800.0;
   stations.current[0].presetTime.critical[7] := 300.0;
   stations.current[0].presetTime.critical[3] := 300.0;
   stations.current[0].partNumbers[7] := WSTRING#'16.32.112.500.100A';
   stations.current[0].partNumbers[6] := WSTRING#'';
   stations.current[0].partNumbers[5] := WSTRING#'';
   stations.current[0].partNumbers[3] := WSTRING#'16.32.112.500.220A';
   stations.current[0].partNumbers[2] := WSTRING#'';
   stations.current[0].partNumbers[1] := WSTRING#'';
   stations.current[0].line := WSTRING#'VOLVO 16';
   stations.current[1].line := WSTRING#'VOLVO 16';
   stations.current[2].line := WSTRING#'VOLVO 16';
   stations.current[0].dropZone := 1;
   stations.current[1].dropZone := 2;
   stations.current[2].dropZone := 3;
   stations.current[3].dropZone := 4;
   stations.current[3].line := WSTRING#'VOLVO 16';
   stations.current[4].dropZone := 5;
   stations.current[4].line := WSTRING#'VOLVO 16';
   stations.current[5].line := WSTRING#'VOLVO 16';
   stations.current[5].dropZone := 6;
   stations.current[6].dropZone := 7;
   stations.current[6].line := WSTRING#'VOLVO 16';
   stations.current[7].dropZone := 8;
   stations.current[7].line := WSTRING#'VOLVO 16';
   stations.current[8].dropZone := 9;
   stations.current[8].line := WSTRING#'VOLVO 16';
   stations.current[9].dropZone := 10;
   stations.current[9].line := WSTRING#'VOLVO 16';
   stations.current[10].dropZone := 11;
   stations.current[10].line := WSTRING#'VOLVO 16';
   stations.current[11].line := WSTRING#'CHM';
   stations.current[11].dropZone := 1;
   stations.current[12].line := WSTRING#'CHM';
   stations.current[12].dropZone := 2;
   stations.current[13].line := WSTRING#'CHM';
   stations.current[13].dropZone := 3;
   stations.current[14].dropZone := 4;
   stations.current[14].line := WSTRING#'CHM';
   stations.current[15].line := WSTRING#'CHM';
   stations.current[15].dropZone := 5;
   stations.current[16].dropZone := 1;
   stations.current[16].line := WSTRING#'CDO';
   stations.current[17].dropZone := 2;
   stations.current[17].line := WSTRING#'CDO';
   stations.current[18].line := WSTRING#'CDO';
   stations.current[18].dropZone := 3;
   stations.current[19].dropZone := 1;
   stations.current[19].line := WSTRING#'BFL';
   stations.current[20].dropZone := 2;
   stations.current[20].line := WSTRING#'BFL';
   stations.current[21].line := WSTRING#'BFL';
   stations.current[21].dropZone := 3;
   stations.current[22].dropZone := 1;
   stations.current[22].line := WSTRING#'LGS';
   stations.current[22].partNumbers[7] := WSTRING#'16.08.216.161.020A';
   stations.current[21].partNumbers[5] := WSTRING#'';
   stations.current[21].partNumbers[6] := WSTRING#'';
   stations.current[21].partNumbers[7] := WSTRING#'16.08.208.011.010G';
   stations.current[18].partNumbers[3] := WSTRING#'16.08.216.911.040B$L16.08.216.200.050A';
   stations.current[18].partNumbers[4] := WSTRING#'';
   stations.current[18].partNumbers[5] := WSTRING#'';
   stations.current[18].partNumbers[6] := WSTRING#'16.08.216.181.020A$L16.08.208.331.000F';
   stations.current[18].partNumbers[7] := WSTRING#'16.08.216.951.010A';
   stations.current[19].partNumbers[7] := WSTRING#'16.08.211.511.020F';
   stations.current[11].partNumbers[0] := WSTRING#'';
   stations.current[11].partNumbers[1] := WSTRING#'';
   stations.current[11].partNumbers[2] := WSTRING#'';
   stations.current[11].partNumbers[3] := WSTRING#'16.08.216.515.008C';
   stations.current[11].partNumbers[4] := WSTRING#'';
   stations.current[11].partNumbers[5] := WSTRING#'';
   stations.current[11].partNumbers[6] := WSTRING#'';
   stations.current[11].partNumbers[7] := WSTRING#'16.08.208.131.010L';
   stations.current[13].partNumbers[0] := WSTRING#'';
   stations.current[13].partNumbers[1] := WSTRING#'';
   stations.current[13].partNumbers[2] := WSTRING#'16.08.216.251.000B';
   stations.current[13].partNumbers[3] := WSTRING#'16.08.216.911.000G';
   stations.current[13].partNumbers[4] := WSTRING#'';
   stations.current[13].partNumbers[5] := WSTRING#'';
   stations.current[13].partNumbers[6] := WSTRING#'16.08.216.911.000H';
   stations.current[13].partNumbers[7] := WSTRING#'16.08.216.911.000C';
   stations.current[14].partNumbers[0] := WSTRING#'';
   stations.current[14].partNumbers[1] := WSTRING#'';
   stations.current[14].partNumbers[2] := WSTRING#'16.08.216.181.100A';
   stations.current[14].partNumbers[3] := WSTRING#'16.08.216.910.020B';
   stations.current[14].partNumbers[4] := WSTRING#'';
   stations.current[14].partNumbers[5] := WSTRING#'16.08.216.181.090A';
   stations.current[14].partNumbers[6] := WSTRING#'16.08.216.722.001A';
   stations.current[14].partNumbers[7] := WSTRING#'16.08.216.181.010B';
   stations.current[18].partNumbers[0] := WSTRING#'';
   stations.current[18].partNumbers[1] := WSTRING#'';
   stations.current[18].partNumbers[2] := WSTRING#'';
   stations.current[12].partNumbers[0] := WSTRING#'';
   stations.current[12].partNumbers[1] := WSTRING#'16.08.216.526.009A';
   stations.current[12].partNumbers[2] := WSTRING#'16.08.216.871.010C';
   stations.current[12].partNumbers[3] := WSTRING#'16.08.216.141.010C';
   stations.current[12].partNumbers[4] := WSTRING#'';
   stations.current[12].partNumbers[5] := WSTRING#'16.08.216.526.002C';
   stations.current[12].partNumbers[6] := WSTRING#'16.08.215.871.010C';
   stations.current[12].partNumbers[7] := WSTRING#'16.08.215.141.010C';
   stations.current[17].partNumbers[0] := WSTRING#'';
   stations.current[17].partNumbers[1] := WSTRING#'';
   stations.current[17].partNumbers[2] := WSTRING#'16.08.216.501.010A';
   stations.current[17].partNumbers[3] := WSTRING#'16.08.208.691.010D';
   stations.current[17].partNumbers[4] := WSTRING#'';
   stations.current[17].partNumbers[5] := WSTRING#'';
   stations.current[17].partNumbers[6] := WSTRING#'16.08.216.790.001A';
   stations.current[17].partNumbers[7] := WSTRING#'16.08.208.531.020L';
   stations.current[15].partNumbers[0] := WSTRING#'';
   stations.current[15].partNumbers[1] := WSTRING#'';
   stations.current[15].partNumbers[2] := WSTRING#'16.08.216.511.000C';
   stations.current[15].partNumbers[3] := WSTRING#'16.08.208.501.000B';
   stations.current[15].partNumbers[4] := WSTRING#'';
   stations.current[15].partNumbers[5] := WSTRING#'16.08.216.551.000B';
   stations.current[15].partNumbers[6] := WSTRING#'16.08.216.231.000B';
   stations.current[15].partNumbers[7] := WSTRING#'16.08.216.501.000C';
   stations.current[16].partNumbers[0] := WSTRING#'';
   stations.current[16].partNumbers[1] := WSTRING#'';
   stations.current[16].partNumbers[2] := WSTRING#'';
   stations.current[16].partNumbers[3] := WSTRING#'16.08.216.912.060B$L16.08.216.202.080A';
   stations.current[16].partNumbers[4] := WSTRING#'';
   stations.current[16].partNumbers[5] := WSTRING#'';
   stations.current[16].partNumbers[6] := WSTRING#'16.08.216.911.030B';
   stations.current[16].partNumbers[7] := WSTRING#'16.08.216.912.050A';
   stations.current[21].partNumbers[0] := WSTRING#'';
   stations.current[21].partNumbers[1] := WSTRING#'';
   stations.current[21].partNumbers[2] := WSTRING#'';
   stations.current[21].partNumbers[3] := WSTRING#'';
   stations.current[21].partNumbers[4] := WSTRING#'';
   stations.current[20].partNumbers[0] := WSTRING#'';
   stations.current[20].partNumbers[1] := WSTRING#'';
   stations.current[20].partNumbers[2] := WSTRING#'';
   stations.current[20].partNumbers[3] := WSTRING#'';
   stations.current[20].partNumbers[4] := WSTRING#'';
   stations.current[20].partNumbers[5] := WSTRING#'';
   stations.current[20].partNumbers[6] := WSTRING#'';
   stations.current[20].partNumbers[7] := WSTRING#'PEANUTS';
   stations.current[8].partNumbers[0] := WSTRING#'';
   stations.current[8].partNumbers[1] := WSTRING#'';
   stations.current[8].partNumbers[2] := WSTRING#'';
   stations.current[8].partNumbers[3] := WSTRING#'16.32.112.580.020A';
   stations.current[8].partNumbers[4] := WSTRING#'';
   stations.current[8].partNumbers[5] := WSTRING#'';
   stations.current[8].partNumbers[6] := WSTRING#'16.32.112.500.300E';
   stations.current[8].partNumbers[7] := WSTRING#'16.32.112.520.300E';
   stations.current[9].partNumbers[0] := WSTRING#'';
   stations.current[9].partNumbers[1] := WSTRING#'';
   stations.current[9].partNumbers[2] := WSTRING#'';
   stations.current[9].partNumbers[3] := WSTRING#'16.32.112.594.000C';
   stations.current[9].partNumbers[4] := WSTRING#'';
   stations.current[9].partNumbers[5] := WSTRING#'';
   stations.current[9].partNumbers[6] := WSTRING#'';
   stations.current[9].partNumbers[7] := WSTRING#'16.32.112.584.000C';
   stations.current[10].partNumbers[0] := WSTRING#'';
   stations.current[10].partNumbers[1] := WSTRING#'';
   stations.current[10].partNumbers[2] := WSTRING#'';
   stations.current[10].partNumbers[3] := WSTRING#'16.32.112.500.150B';
   stations.current[10].partNumbers[4] := WSTRING#'';
   stations.current[10].partNumbers[5] := WSTRING#'';
   stations.current[10].partNumbers[6] := WSTRING#'16.32.806.502.080A';
   stations.current[10].partNumbers[7] := WSTRING#'16.32.112.500.160A';
   stations.current[0].partNumbers[0] := WSTRING#'';
   stations.current[0].partNumbers[4] := WSTRING#'';
   stations.current[1].partNumbers[0] := WSTRING#'';
   stations.current[1].partNumbers[1] := WSTRING#'';
   stations.current[1].partNumbers[2] := WSTRING#'16.32.112.509.070A';
   stations.current[1].partNumbers[3] := WSTRING#'16.32.112.704.000C';
   stations.current[1].partNumbers[4] := WSTRING#'';
   stations.current[1].partNumbers[5] := WSTRING#'';
   stations.current[1].partNumbers[6] := WSTRING#'16.32.112.504.060A';
   stations.current[1].partNumbers[7] := WSTRING#'16.32.112.500.060D';
   stations.current[2].partNumbers[0] := WSTRING#'';
   stations.current[2].partNumbers[1] := WSTRING#'16.32.112.509.050E';
   stations.current[2].partNumbers[2] := WSTRING#'16.32.112.504.070G';
   stations.current[2].partNumbers[3] := WSTRING#'16.32.112.851.001A';
   stations.current[2].partNumbers[4] := WSTRING#'';
   stations.current[2].partNumbers[5] := WSTRING#'16.32.112.509.080F';
   stations.current[2].partNumbers[6] := WSTRING#'16.32.112.870.000C';
   stations.current[2].partNumbers[7] := WSTRING#'16.32.112.851.000A';
   stations.current[3].partNumbers[0] := WSTRING#'';
   stations.current[3].partNumbers[1] := WSTRING#'16.32.112.522.130A';
   stations.current[3].partNumbers[2] := WSTRING#'16.32.112.522.050A';
   stations.current[3].partNumbers[3] := WSTRING#'16.32.112.521.020B';
   stations.current[3].partNumbers[4] := WSTRING#'';
   stations.current[3].partNumbers[5] := WSTRING#'16.32.112.522.040D';
   stations.current[3].partNumbers[6] := WSTRING#'16.32.112.521.010B';
   stations.current[3].partNumbers[7] := WSTRING#'16.32.112.521.030A';
   stations.current[4].partNumbers[0] := WSTRING#'';
   stations.current[4].partNumbers[1] := WSTRING#'';
   stations.current[4].partNumbers[2] := WSTRING#'';
   stations.current[4].partNumbers[3] := WSTRING#'';
   stations.current[4].partNumbers[4] := WSTRING#'';
   stations.current[4].partNumbers[5] := WSTRING#'';
   stations.current[4].partNumbers[6] := WSTRING#'';
   stations.current[4].partNumbers[7] := WSTRING#'16.32.112.529.020B';
   stations.current[5].partNumbers[0] := WSTRING#'';
   stations.current[5].partNumbers[1] := WSTRING#'16.32.112.529.010A';
   stations.current[5].partNumbers[2] := WSTRING#'16.32.112.529.030A';
   stations.current[5].partNumbers[3] := WSTRING#'16.32.112.502.060B';
   stations.current[5].partNumbers[4] := WSTRING#'';
   stations.current[5].partNumbers[5] := WSTRING#'16.32.112.529.050D';
   stations.current[5].partNumbers[6] := WSTRING#'16.32.112.502.070E';
   stations.current[5].partNumbers[7] := WSTRING#'16.32.112.502.050B';
   stations.current[6].partNumbers[0] := WSTRING#'';
   stations.current[6].partNumbers[1] := WSTRING#'16.32.112.621.020A';
   stations.current[6].partNumbers[2] := WSTRING#'16.32.112.621.010A';
   stations.current[6].partNumbers[3] := WSTRING#'16.32.112.751.000D';
   stations.current[6].partNumbers[4] := WSTRING#'';
   stations.current[6].partNumbers[5] := WSTRING#'16.32.112.751.001C';
   stations.current[6].partNumbers[6] := WSTRING#'16.32.112.601.040A';
   stations.current[6].partNumbers[7] := WSTRING#'16.32.112.601.030A';
   stations.current[7].partNumbers[0] := WSTRING#'';
   stations.current[7].partNumbers[1] := WSTRING#'';
   stations.current[7].partNumbers[2] := WSTRING#'';
   stations.current[7].partNumbers[3] := WSTRING#'16.32.112.500.520B';
   stations.current[7].partNumbers[4] := WSTRING#'';
   stations.current[7].partNumbers[5] := WSTRING#'';
   stations.current[7].partNumbers[6] := WSTRING#'16.32.112.500.090B';
   stations.current[7].partNumbers[7] := WSTRING#'16.32.112.500.120A';
   stations.current[23].line := WSTRING#'LGS';
   stations.current[23].dropZone := 2;
   stations.current[23].partNumbers[0] := WSTRING#'';
   stations.current[23].partNumbers[1] := WSTRING#'';
   stations.current[23].partNumbers[2] := WSTRING#'';
   stations.current[23].partNumbers[3] := WSTRING#'';
   stations.current[23].partNumbers[4] := WSTRING#'';
   stations.current[23].partNumbers[5] := WSTRING#'';
   stations.current[23].partNumbers[6] := WSTRING#'';
   stations.current[23].partNumbers[7] := WSTRING#'16.08.208.021.020C';
   stations.current[22].partNumbers[0] := WSTRING#'';
   stations.current[22].partNumbers[1] := WSTRING#'';
   stations.current[22].partNumbers[2] := WSTRING#'';
   stations.current[22].partNumbers[3] := WSTRING#'16.08.208.161.020F';
   stations.current[22].partNumbers[4] := WSTRING#'';
   stations.current[22].partNumbers[5] := WSTRING#'';
   stations.current[22].partNumbers[6] := WSTRING#'OP60 - STAMPINGS';
   stations.current[19].partNumbers[0] := WSTRING#'';
   stations.current[19].partNumbers[1] := WSTRING#'';
   stations.current[19].partNumbers[2] := WSTRING#'16.08.216.831.020A';
   stations.current[19].partNumbers[3] := WSTRING#'16.08.208.151.010F';
   stations.current[19].partNumbers[4] := WSTRING#'';
   stations.current[19].partNumbers[5] := WSTRING#'16.08.217.411.080A';
   stations.current[19].partNumbers[6] := WSTRING#'16.08.216.151.010B';
   constants.hmiRowCount := 12;
END_DATA_BLOCK

DATA_BLOCK "HMI"   // DB2
{ S7_Optimized_Access := 'TRUE' }
VERSION : 0.1
   VAR
      partCall : "Part Call Screen";
      screenNumber : Int;
      settings : "Settings Screen";
      barcode : "Barcode Screen";
   END_VAR
BEGIN
   settings.current.kp8.buttons[1].label := WSTRING#'6';
   settings.current.kp8.buttons[2].label := WSTRING#'4';
   settings.current.kp8.buttons[3].label := WSTRING#'2';
   settings.current.kp8.buttons[5].label := WSTRING#'5';
   settings.current.kp8.buttons[6].label := WSTRING#'3';
   settings.current.kp8.buttons[7].label := WSTRING#'1';
END_DATA_BLOCK

DATA_BLOCK "Parts"   // DB3
{ S7_Optimized_Access := 'TRUE' }
VERSION : 0.1
   VAR
      pRow : Int;
   END_VAR
   VAR RETAIN
      requests : "Part Request Data";
   END_VAR
BEGIN
END_DATA_BLOCK

DATA_BLOCK "LED Sign"   // DB4
{ S7_Optimized_Access := 'TRUE' }
VERSION : 0.1
   VAR
      request : "LED Sign Data";
   END_VAR
BEGIN
END_DATA_BLOCK

FUNCTION_BLOCK "EMP"   // FB1, LAD
{ S7_Optimized_Access := 'TRUE' }
VERSION : 0.1
   VAR RETAIN
      constants : "Constants";
   END_VAR
   VAR
      instBaseAnimations : "Base Animations";
      instHMIAnimations : "Format Part Call Requests";
      instInitialize : "Initialize";
      instKP8ButtonActivation : "KP8 Button Activation";
      instKP8ExpandedAnimations : "KP8 Expanded Animations";
      instPartTimers : "Part Timers";
      instRecordPartRequest : "Record Part Request";
      instRemovePartRequest : "Remove Part Request";
      instResetInitRequest : "Reset Init Requests";
      instStackLightAnimations : "Stack Light Animations";
      "KP8 Drivers" : Array[0..#stationCount] of "KP8 Driver";
   END_VAR
   VAR RETAIN
      stations : "Stations";
   END_VAR
   VAR
      instHMIBarcode : "HMI Barcod Screen";
      instCollapseTable : "Collapse Table";
      instPopulateHMI : "HMI Populate Part Call";
      instHMISettings : "HMI Settings Screen";
      instClearReqData : "Clear Part Requests";
      instDefaultTmrPrst : "Load Default Timer Presets";
      instPopulateLED : "LED Populate Sign";
   END_VAR
   VAR_TEMP
      i : Int;
      stnCount : Int;
   END_VAR
   VAR CONSTANT
      stationCount : Int := 24;
   END_VAR
BEGIN

REGION Network 1: PHYSICAL TO GLOBAL
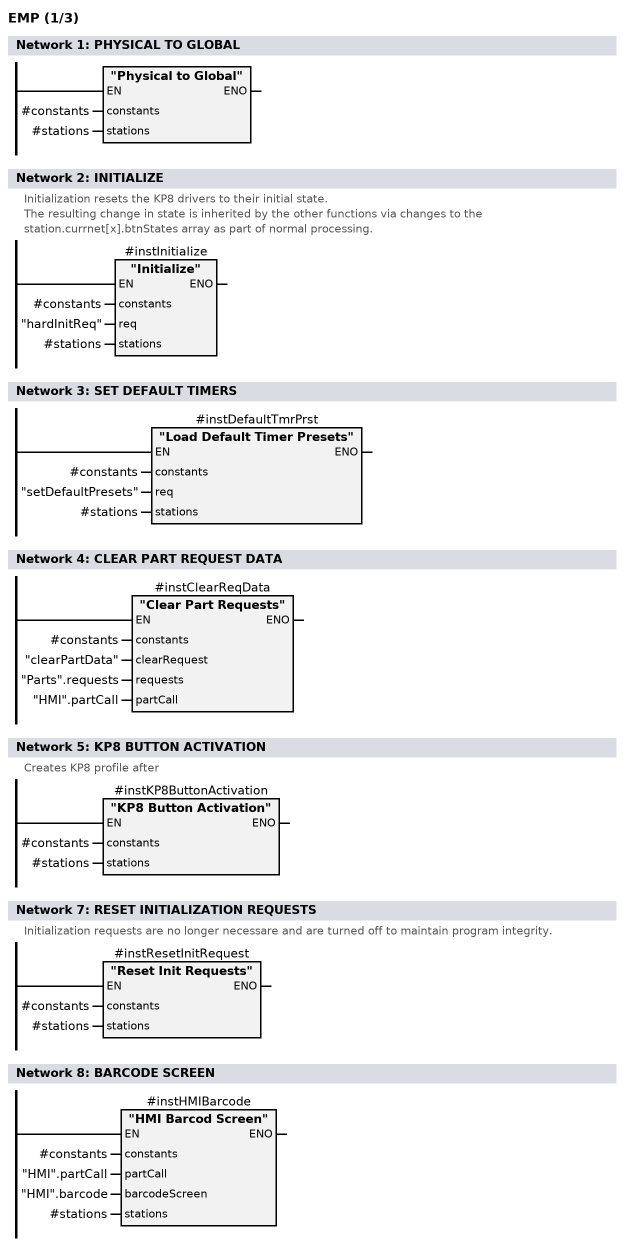
   RUNG wire#powerrail
      "Physical to Global"(constants := #constants, stations := #stations)
   END_RUNG
   // the same network as SCL:
   "Physical to Global"(constants := #constants, stations := #stations);
END_REGION

REGION Network 2: INITIALIZE
   // Initialization resets the KP8 drivers to their initial state.
   // The resulting change in state is inherited by the other functions via changes to the
   // station.currnet[x].btnStates array as part of normal processing.
   RUNG wire#powerrail
      #instInitialize(constants := #constants, req := "hardInitReq", stations := #stations)
   END_RUNG
   // the same network as SCL:
   #instInitialize(constants := #constants, req := "hardInitReq", stations := #stations);   // "Initialize"
END_REGION

REGION Network 3: SET DEFAULT TIMERS
   RUNG wire#powerrail
      #instDefaultTmrPrst(constants := #constants, req := "setDefaultPresets", stations := #stations)
   END_RUNG
   // the same network as SCL:
   #instDefaultTmrPrst(constants := #constants, req := "setDefaultPresets", stations := #stations);   // "Load Default Timer Presets"
END_REGION

REGION Network 4: CLEAR PART REQUEST DATA
   RUNG wire#powerrail
      #instClearReqData(constants := #constants, clearRequest := "clearPartData", requests := "Parts".requests, partCall := "HMI".partCall)
   END_RUNG
   // the same network as SCL:
   #instClearReqData(constants := #constants,   // "Clear Part Requests"
                     clearRequest := "clearPartData",
                     requests := "Parts".requests,
                     partCall := "HMI".partCall);
END_REGION

REGION Network 5: KP8 BUTTON ACTIVATION
   // Creates KP8 profile after
   RUNG wire#powerrail
      #instKP8ButtonActivation(constants := #constants, stations := #stations)
   END_RUNG
   // the same network as SCL:
   #instKP8ButtonActivation(constants := #constants, stations := #stations);   // "KP8 Button Activation"
END_REGION

REGION Network 6 (SCL): KP8 DRIVER CALLS
   REGION "LOOP THROUGH STATIONS"
       #stnCount := #constants.stationCount - 1;
       FOR #i := 0 TO #stnCount DO
           #"KP8 Drivers"[#i](btnIn := #stations.current[#i].kp8In,
                              hardInit := #stations.current[#i].init.hard,
                              softInit := #stations.current[#i].init.soft,
                              btn0Activate := #stations.current[#i].kp8Config.activate[0],
                              btn0Mode := #stations.current[#i].kp8Config.mode[0],
                              btn0Group := #stations.current[#i].kp8Config.group[0],
                              btn0Flash := #stations.current[#i].kp8Config.flash[0],
                              btn0ColorOn1 := #stations.current[#i].kp8Config.colorOn1[0],
                              btn0ColorOn2 := #stations.current[#i].kp8Config.colorOn2[0],
                              btn0ColorOff := #stations.current[#i].kp8Config.colorOff[0],
                              btn1Activate := #stations.current[#i].kp8Config.activate[1],
                              btn1Mode := #stations.current[#i].kp8Config.mode[1],
                              btn1Group := #stations.current[#i].kp8Config.group[1],
                              btn1Flash := #stations.current[#i].kp8Config.flash[1],
                              btn1ColorOn1 := #stations.current[#i].kp8Config.colorOn1[1],
                              btn1ColorOn2 := #stations.current[#i].kp8Config.colorOn2[1],
                              btn1ColorOff := #stations.current[#i].kp8Config.colorOff[1],
                              btn2Activate := #stations.current[#i].kp8Config.activate[2],
                              btn2Mode := #stations.current[#i].kp8Config.mode[2],
                              btn2Group := #stations.current[#i].kp8Config.group[2],
                              btn2Flash := #stations.current[#i].kp8Config.flash[2],
                              btn2ColorOn1 := #stations.current[#i].kp8Config.colorOn1[2],
                              btn2ColorOn2 := #stations.current[#i].kp8Config.colorOn2[2],
                              btn2ColorOff := #stations.current[#i].kp8Config.colorOff[2],
                              btn3Activate := #stations.current[#i].kp8Config.activate[3],
                              btn3Mode := #stations.current[#i].kp8Config.mode[3],
                              btn3Group := #stations.current[#i].kp8Config.group[3],
                              btn3Flash := #stations.current[#i].kp8Config.flash[3],
                              btn3ColorOn1 := #stations.current[#i].kp8Config.colorOn1[3],
                              btn3ColorOn2 := #stations.current[#i].kp8Config.colorOn2[3],
                              btn3ColorOff := #stations.current[#i].kp8Config.colorOff[3],
                              btn4Activate := #stations.current[#i].kp8Config.activate[4],
                              btn4Mode := #stations.current[#i].kp8Config.mode[4],
                              btn4Group := #stations.current[#i].kp8Config.group[4],
                              btn4Flash := #stations.current[#i].kp8Config.flash[4],
                              btn4ColorOn1 := #stations.current[#i].kp8Config.colorOn1[4],
                              btn4ColorOn2 := #stations.current[#i].kp8Config.colorOn2[4],
                              btn4ColorOff := #stations.current[#i].kp8Config.colorOff[4],
                              btn5Activate := #stations.current[#i].kp8Config.activate[5],
                              btn5Mode := #stations.current[#i].kp8Config.mode[5],
                              btn5Group := #stations.current[#i].kp8Config.group[5],
                              btn5Flash := #stations.current[#i].kp8Config.flash[5],
                              btn5ColorOn1 := #stations.current[#i].kp8Config.colorOn1[5],
                              btn5ColorOn2 := #stations.current[#i].kp8Config.colorOn2[5],
                              btn5ColorOff := #stations.current[#i].kp8Config.colorOff[5],
                              btn6Activate := #stations.current[#i].kp8Config.activate[6],
                              btn6Mode := #stations.current[#i].kp8Config.mode[6],
                              btn6Group := #stations.current[#i].kp8Config.group[6],
                              btn6Flash := #stations.current[#i].kp8Config.flash[6],
                              btn6ColorOn1 := #stations.current[#i].kp8Config.colorOn1[6],
                              btn6ColorOn2 := #stations.current[#i].kp8Config.colorOn2[6],
                              btn6ColorOff := #stations.current[#i].kp8Config.colorOff[6],
                              btn7Activate := #stations.current[#i].kp8Config.activate[7],
                              btn7Mode := #stations.current[#i].kp8Config.mode[7],
                              btn7Group := #stations.current[#i].kp8Config.group[7],
                              btn7Flash := #stations.current[#i].kp8Config.flash[7],
                              btn7ColorOn1 := #stations.current[#i].kp8Config.colorOn1[7],
                              btn7ColorOn2 := #stations.current[#i].kp8Config.colorOn2[7],
                              btn7ColorOff := #stations.current[#i].kp8Config.colorOff[7],
                              btnStatesOut => #stations.current[#i].btnStates,
                              btnColorsOut => #stations.current[#i].kp8Out);
       END_FOR;
   END_REGION
END_REGION

REGION Network 7: RESET INITIALIZATION REQUESTS
   // Initialization requests are no longer necessare and are turned off to maintain program integrity.
   RUNG wire#powerrail
      #instResetInitRequest(constants := #constants, stations := #stations)
   END_RUNG
   // the same network as SCL:
   #instResetInitRequest(constants := #constants, stations := #stations);   // "Reset Init Requests"
END_REGION

REGION Network 8: BARCODE SCREEN
   RUNG wire#powerrail
      #instHMIBarcode(constants := #constants, partCall := "HMI".partCall, barcodeScreen := "HMI".barcode, stations := #stations)
   END_RUNG
   // the same network as SCL:
   #instHMIBarcode(constants := #constants,   // "HMI Barcod Screen"
                   partCall := "HMI".partCall,
                   barcodeScreen := "HMI".barcode,
                   stations := #stations);
END_REGION

REGION Network 9: PART TIMERS
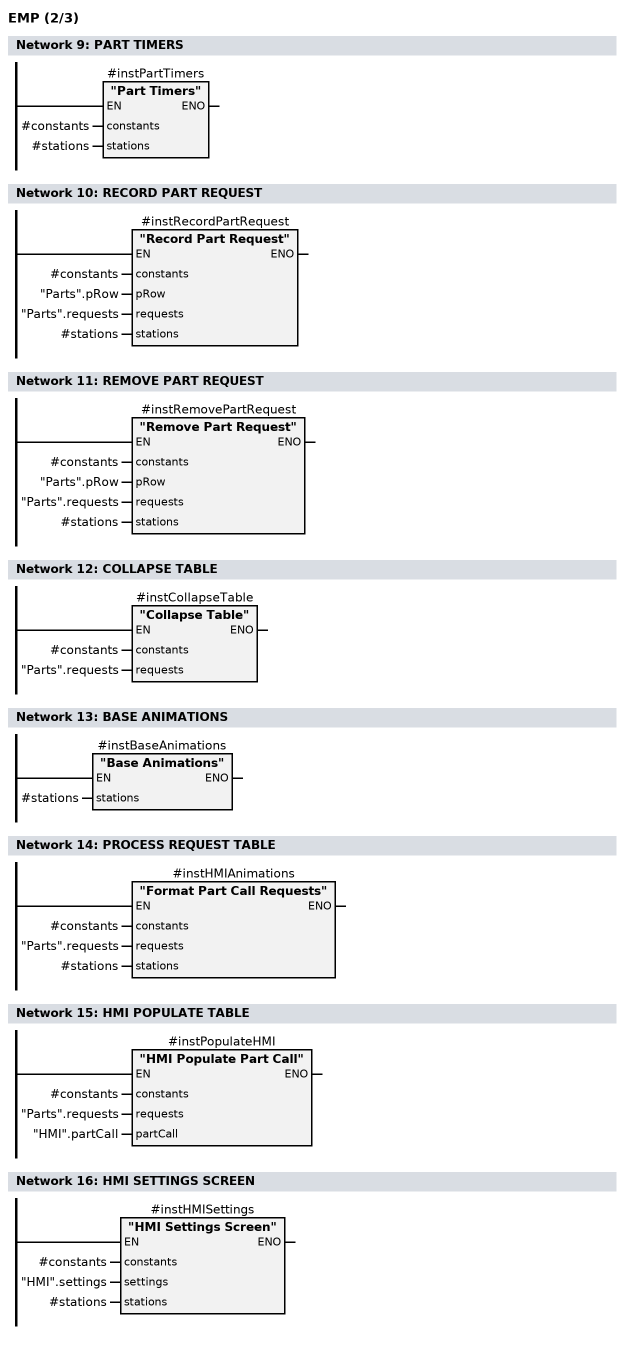
   RUNG wire#powerrail
      #instPartTimers(constants := #constants, stations := #stations)
   END_RUNG
   // the same network as SCL:
   #instPartTimers(constants := #constants, stations := #stations);   // "Part Timers"
END_REGION

REGION Network 10: RECORD PART REQUEST
   RUNG wire#powerrail
      #instRecordPartRequest(constants := #constants, pRow := "Parts".pRow, requests := "Parts".requests, stations := #stations)
   END_RUNG
   // the same network as SCL:
   #instRecordPartRequest(constants := #constants,   // "Record Part Request"
                          pRow := "Parts".pRow,
                          requests := "Parts".requests,
                          stations := #stations);
END_REGION

REGION Network 11: REMOVE PART REQUEST
   RUNG wire#powerrail
      #instRemovePartRequest(constants := #constants, pRow := "Parts".pRow, requests := "Parts".requests, stations := #stations)
   END_RUNG
   // the same network as SCL:
   #instRemovePartRequest(constants := #constants,   // "Remove Part Request"
                          pRow := "Parts".pRow,
                          requests := "Parts".requests,
                          stations := #stations);
END_REGION

REGION Network 12: COLLAPSE TABLE
   RUNG wire#powerrail
      #instCollapseTable(constants := #constants, requests := "Parts".requests)
   END_RUNG
   // the same network as SCL:
   #instCollapseTable(constants := #constants, requests := "Parts".requests);   // "Collapse Table"
END_REGION

REGION Network 13: BASE ANIMATIONS
   RUNG wire#powerrail
      #instBaseAnimations(stations := #stations)
   END_RUNG
   // the same network as SCL:
   #instBaseAnimations(stations := #stations);   // "Base Animations"
END_REGION

REGION Network 14: PROCESS REQUEST TABLE
   RUNG wire#powerrail
      #instHMIAnimations(constants := #constants, requests := "Parts".requests, stations := #stations)
   END_RUNG
   // the same network as SCL:
   #instHMIAnimations(constants := #constants, requests := "Parts".requests, stations := #stations);   // "Format Part Call Requests"
END_REGION

REGION Network 15: HMI POPULATE TABLE
   RUNG wire#powerrail
      #instPopulateHMI(constants := #constants, requests := "Parts".requests, partCall := "HMI".partCall)
   END_RUNG
   // the same network as SCL:
   #instPopulateHMI(constants := #constants, requests := "Parts".requests, partCall := "HMI".partCall);   // "HMI Populate Part Call"
END_REGION

REGION Network 16: HMI SETTINGS SCREEN
   RUNG wire#powerrail
      #instHMISettings(constants := #constants, settings := "HMI".settings, stations := #stations)
   END_RUNG
   // the same network as SCL:
   #instHMISettings(constants := #constants, settings := "HMI".settings, stations := #stations);   // "HMI Settings Screen"
END_REGION

REGION Network 17: LED POPULATE SIGN
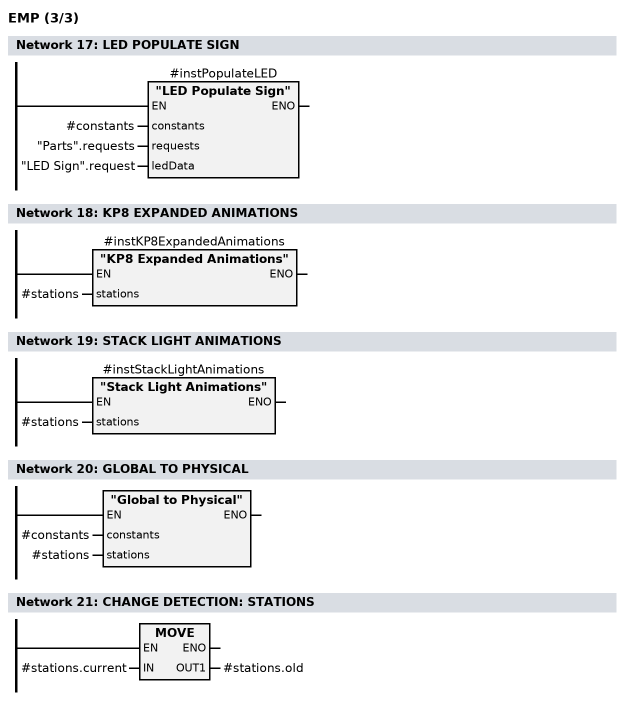
   RUNG wire#powerrail
      #instPopulateLED(constants := #constants, requests := "Parts".requests, ledData := "LED Sign".request)
   END_RUNG
   // the same network as SCL:
   #instPopulateLED(constants := #constants, requests := "Parts".requests, ledData := "LED Sign".request);   // "LED Populate Sign"
END_REGION

REGION Network 18: KP8 EXPANDED ANIMATIONS
   RUNG wire#powerrail
      #instKP8ExpandedAnimations(stations := #stations)
   END_RUNG
   // the same network as SCL:
   #instKP8ExpandedAnimations(stations := #stations);   // "KP8 Expanded Animations"
END_REGION

REGION Network 19: STACK LIGHT ANIMATIONS
   RUNG wire#powerrail
      #instStackLightAnimations(stations := #stations)
   END_RUNG
   // the same network as SCL:
   #instStackLightAnimations(stations := #stations);   // "Stack Light Animations"
END_REGION

REGION Network 20: GLOBAL TO PHYSICAL
   RUNG wire#powerrail
      "Global to Physical"(constants := #constants, stations := #stations)
   END_RUNG
   // the same network as SCL:
   "Global to Physical"(constants := #constants, stations := #stations);
END_REGION

REGION Network 21: CHANGE DETECTION: STATIONS
   RUNG wire#powerrail
      Move(in := #stations.current, out1 => #stations.old)
   END_RUNG
   // the same network as SCL:
   #stations.old := #stations.current;
END_REGION
END_FUNCTION_BLOCK

FUNCTION_BLOCK "Code 128"   // FB2, SCL
{ S7_Optimized_Access := 'TRUE' }
VERSION : 0.1
   VAR_INPUT
      partNumber : String;
   END_VAR
   VAR_OUTPUT
      barcode : String;
   END_VAR
   VAR
      charsIn : Array[0..255] of Byte;
      charsOut : Array[0..255] of Byte;
      cnt : UInt;
      intVals : Array[0..255] of Int;
      sum : Int;
      checkSum : Int;
   END_VAR
   VAR_TEMP
      pn : String;
      i : Int;
   END_VAR
   VAR CONSTANT
      startChar : Char := 'Ì';
      stopChar : Char := 'Î';
   END_VAR
   // intVals[0] := 104;
BEGIN
   #pn := #partNumber;

   FOR #i := 0 TO 255 DO
       #charsIn[#i] := 16#00;
       #charsOut[#i] := 16#00;
       #intVals[#i] := 0;
   END_FOR;

   Strg_TO_Chars(Strg:=#pn,
                 pChars:=0,
                 Cnt=>#cnt,
                 Chars:=#charsIn);


   #sum := 104;
   FOR #i := 0 TO UINT_TO_INT(#cnt - 1) DO
       #intVals[#i] := CHAR_TO_INT(#charsIn[#i]) - 32;
       #intVals[#i] := #intVals[#i] * (#i + 1);
       #sum := #sum + #intVals[#i];
   END_FOR;
   #checkSum := (#sum MOD 103) + 32;
   IF #checkSum >= 127 THEN
       #checkSum := #checkSum + 68;
   END_IF;

   #charsOut[0] := #startChar;
   FOR #i := 1 TO UINT_TO_INT(#cnt) DO
       #charsOut[#i] := #charsIn[#i - 1];
   END_FOR;
   #charsOut[#cnt + 1] := INT_TO_BYTE(#checkSum);
   #charsOut[#cnt + 2] := INT_TO_BYTE(#stopChar);

   Chars_TO_Strg(Chars := #charsOut,
                 pChars := 0,
                 Cnt := #cnt + 3,
                 Strg => #barcode);
END_FUNCTION_BLOCK

FUNCTION_BLOCK "HMI Barcod Screen"   // FB3, SCL
{ S7_Optimized_Access := 'TRUE' }
VERSION : 0.1
   VAR_INPUT
      constants : "Constants";
   END_VAR
   VAR_IN_OUT
      partCall : "Part Call Screen";
      barcodeScreen : "Barcode Screen";
      stations : "Stations";
   END_VAR
   VAR
      address : UInt;
      button : UInt;
      instCode128 : "Code 128";
      codeOut : String;
      pnOut : WString[40];
      station : UInt;
      oldSelectedRow : Int;
   END_VAR
   VAR_TEMP
      orderCancelled : Int;
      processedPN : String[40];
      selectedPN : String[40];
      userOrdered : Bool;
      selectedRow : Int;
   END_VAR
   VAR CONSTANT
      maxRows : Int := 199;
   END_VAR
BEGIN
   REGION "GET USER ROW SELECTION"
       #selectedRow := "Get Part Call Row Number"(constants := #constants,
                                                  partCall := #partCall);
   END_REGION

   REGION "ON SELECTION OF A PART CALL ROW
       IF #selectedRow <> 0 THEN
           IF #selectedRow <> #oldSelectedRow THEN

               REGION "GET BUTTON AND STATION NUMBERS"
                   #address := #partCall.current[#selectedRow - 1].address;
                   "Address to Station and Button"(address := #address,
                                                   station => #station,
                                                   button => #button);
               END_REGION

               REGION "CONVERT STRING TO BARCODE"

                   REGION "COPY TO LOCALS"
                       #selectedPN := WSTRING_TO_STRING(#partCall.current[#selectedRow - 1].tfPartNumber.value);
                   END_REGION

                   REGION "CONVERT TO BARCODE"
                       #instCode128(partNumber := #processedPN,
                                    barcode => #codeOut);
                   END_REGION

                   REGION "OUTPUT FOR HMI SCREEN"
                       #barcodeScreen.partNumber := STRING_TO_WSTRING(#processedPN);
                       #barcodeScreen.barcode := #codeOut;
                   END_REGION

               END_REGION

           END_IF;
       END_IF;
   END_REGION

   REGION "PASS USER ORDERED"
       // get input
       #userOrdered := #barcodeScreen.ordered;
       // put into station
       #stations.current[#station].partOrdered[#button] := #userOrdered;
   END_REGION


   #oldSelectedRow := #selectedRow;
END_FUNCTION_BLOCK

FUNCTION_BLOCK "Initialize"   // FB4, SCL
{ S7_Optimized_Access := 'TRUE' }
VERSION : 0.1
   VAR_INPUT
      constants : "Constants";
      req : Bool;
   END_VAR
   VAR_IN_OUT
      stations : "Stations";
   END_VAR
   VAR
      rtElapsed : Real;
      rt : Struct
         elapsed : LReal;
         mem : LReal;
      END_STRUCT;
   END_VAR
   VAR_TEMP
      i : Int;
      reset : Struct
         req : Bool;
         elapsed : Real;
      END_STRUCT;
      stnCount : Int;
      init : Bool;
   END_VAR
   VAR CONSTANT
      resetLimit : Real := 1.25;
   END_VAR
BEGIN
   REGION "GET STATION COUNT"
       #stnCount := #constants.stationCount - 1;
   END_REGION

   REGION "FIRST SCAN OR REQUEST"
       IF "FirstScan" OR #req THEN
           // initialize all stations on plc first scan
           FOR #i := 0 TO #stnCount DO
               #stations.current[#i].init.hard := TRUE;
           END_FOR;
       END_IF;
   END_REGION

   REGION "RUNTIME CALL"
       // get elapsed time
       #rt.elapsed := RUNTIME(#rt.mem);
       // convert to real data type
       #rtElapsed := LREAL_TO_REAL(#rt.elapsed);
   END_REGION

   REGION "BUTTON 0 BASED RESET TIMERS"
       FOR #i := 0 TO #stnCount DO

           REGION "PRE-CONDITION"
               // init off by default
               #init := FALSE;
               // request is button 0 on kp8
               #reset.req := #stations.current[#i].kp8In.%X0;
               // saved to shorter name
               #reset.elapsed := #stations.current[#i].elapsedTime.resetReq;
           END_REGION

           REGION "RESET REQUEST"
               IF NOT #reset.req THEN
                   #reset.elapsed := 0.0;
               END_IF;
               IF #reset.req THEN
                   // incriment elapsed time
                   #reset.elapsed := #reset.elapsed + #rtElapsed;
                   // timer expired condition
                   IF #reset.elapsed >= #resetLimit THEN
                       #init := TRUE;
                       #reset.elapsed := 0.0;
                   END_IF;
               END_IF;
               // save elapsed time
               #stations.current[#i].elapsedTime.resetReq := #reset.elapsed;
           END_REGION

           REGION "SAVE INITIALIZATIN REQUEST"
               #stations.current[#i].init.hard := #init;
           END_REGION

       END_FOR;
   END_REGION
END_FUNCTION_BLOCK

FUNCTION_BLOCK "Reset Init Requests"   // FB5, SCL
{ S7_Optimized_Access := 'TRUE' }
VERSION : 0.1
   VAR_INPUT
      constants : "Constants";
   END_VAR
   VAR_IN_OUT
      stations : "Stations";
   END_VAR
   VAR
      placeHolder : Bool;
   END_VAR
   VAR_TEMP
      i : Int;
      stnCount : Int;
   END_VAR
BEGIN
   REGION "GET STATION COUNT"
       #stnCount := #constants.stationCount - 1;
   END_REGION

   REGION "RESET INITIALIZATION REQUESTS
       FOR #i := 0 TO #stnCount DO
           #stations.current[#i].init.hard := FALSE;
           #stations.current[#i].init.soft := FALSE;
       END_FOR;
   END_REGION
END_FUNCTION_BLOCK

FUNCTION_BLOCK "Record Part Request"   // FB6, SCL
{ S7_Optimized_Access := 'TRUE' }
VERSION : 0.1
   VAR_INPUT
      constants : "Constants";
   END_VAR
   VAR_IN_OUT
      pRow : Int;
      requests : "Part Request Data";
      stations : "Stations";
   END_VAR
   VAR
      enterAddress : Bool;
   END_VAR
   VAR_TEMP
      address : UInt;
      hasPart : Bool;
      i : Int;
      intTime : Int;
      j : Int;
      k : Int;
      logAddress : UInt;
      noPart : Bool;
      oldPartReq : Bool;
      partReq : Bool;
      partNumber : WString;
      timeTime : Time;
      wstringTime : WString;
      stnCount : Int;
      maxReqRows : Int;
   END_VAR
BEGIN
   REGION "COPY TO LOCAL"
       #maxReqRows := #constants.partReqRows - 1;
       #stnCount := #constants.stationCount - 1;
   END_REGION

   REGION "MAIN LOOP"
       FOR #i := 0 TO #stnCount DO

           REGION "LOOP THROUGH BUTTONS"
               // j = 0 is excluded because it is used as a station reset button
               FOR #j := 1 TO 7 DO

                   REGION "PRE-CONDITION"
                       // bits for new request detection
                       #partReq := #stations.current[#i].btnStates[#j];
                       #oldPartReq := #stations.old[#i].btnStates[#j];
                   END_REGION

                   REGION "DETERMINE STATE"
                       // new request detection
                       IF #partReq AND NOT #oldPartReq THEN
                           // save to local
                           #partNumber := #stations.current[#i].partNumbers[#j];
                           // no part number
                           IF LEN(#partNumber) = 0 THEN
                               #hasPart := FALSE;
                               #noPart := TRUE;
                           END_IF;
                           // has part number
                           IF LEN(#partNumber) <> 0 THEN
                               #hasPart := TRUE;
                               #noPart := FALSE;
                           END_IF;
                       END_IF;
                   END_REGION

                   REGION "NO PART"
                       IF #noPart THEN
                           // turn off the lights
                           #hasPart := FALSE;
                           #noPart := FALSE;
                           #enterAddress := FALSE;
                       END_IF;
                   END_REGION

                   REGION "HAS PART"
                       IF #hasPart THEN
                           // turn off the lights
                           #hasPart := FALSE;
                           // calculate address
                           #address := (INT_TO_UINT(#i) + 1) * 10 + (INT_TO_UINT(#j) + 1);
                           // precondition enter address flag
                           #enterAddress := TRUE;
                           // check table for previous entry
                           FOR #k := 0 TO #maxReqRows DO
                               // save to local
                               #logAddress := #requests.row[#k].address;
                               // do not re-enter previous requests
                               IF #logAddress = #address THEN
                                   #enterAddress := FALSE;
                               END_IF;
                           END_FOR;
                       END_IF;
                   END_REGION

                   REGION "ENTER ADDRESS"
                       IF #enterAddress THEN
                           // turn off the lights
                           #enterAddress := FALSE;
                           // no processing needed
                           #requests.row[#pRow].address := #address;
                           #requests.row[#pRow].tfLine.value := #stations.current[#i].line;
                           // drop zone is unsigned so simple conversion is okay
                           #requests.row[#pRow].tfDropZone.value := USINT_TO_WSTRING(#stations.current[#i].dropZone);
                           // no processing needed
                           #requests.row[#pRow].tfPartNumber.value := #stations.current[#i].partNumbers[#j];
                           // several steps to change real to time based wstring
                           #intTime := REAL_TO_INT(#stations.current[#i].elapsedTime.partReq[#j]);
                           #timeTime := INT_TO_TIME(#intTime);
                           #wstringTime := "Time to WString"(#timeTime);
                           #requests.row[#pRow].tfTime.value := #wstringTime;
                           // incriment row pointer
                           #pRow := #pRow + 1;
                           IF #pRow > #maxReqRows THEN
                               #pRow := 0;
                           END_IF;
                       END_IF;
                   END_REGION

               END_FOR;
           END_REGION

       END_FOR;
   END_REGION
END_FUNCTION_BLOCK

FUNCTION_BLOCK "Part Timers"   // FB7, SCL
{ S7_Optimized_Access := 'TRUE' }
VERSION : 0.1
   VAR_INPUT
      constants : "Constants";
   END_VAR
   VAR_IN_OUT
      stations : "Stations";
   END_VAR
   VAR
      rt : "Runtime Data";
   END_VAR
   VAR_TEMP
      alottedTime : Real;
      btnCount : Int;
      elapsedTime : Real;
      i : Int;
      j : Int;
      partRequested : Bool;
      redTime : Real;
      remainingTime : Real;
      stnCount : Int;
      press : Struct
         current : Bool;
         old : Bool;
      END_STRUCT;
   END_VAR
BEGIN
   REGION "RUNTIME CALL"
       #rt.elapsed := RUNTIME(#rt.mem);
       #rt.asReal := LREAL_TO_REAL(#rt.elapsed);
   END_REGION

   REGION "GET STATION COUNT"
       #stnCount := #constants.stationCount - 1;
       #btnCount := #constants.buttonCount - 1;
   END_REGION

   REGION "MAIN LOOP"
       FOR #i := 0 TO #stnCount DO
           // j := 0 would be the reset button so it is skipped
           FOR #j := 1 TO #btnCount DO

               REGION "RESET PART TIMER"
                   #press.current := #stations.current[#i].btnStates[#j];
                   #press.old := #stations.old[#i].btnStates[#j];
                   IF NOT #press.current AND #press.old THEN
                           #stations.current[#i].elapsedTime.partReq[#j] := 0.0;
                   END_IF;
               END_REGION

               REGION "PART REQUEST TIMER"
                   // get and check button state 
                   #partRequested := #stations.current[#i].btnStates[#j];
                   IF #partRequested THEN

                       REGION "OUTPUT ELLAPSED TIME"
                           // get saved time
                           #elapsedTime := #stations.current[#i].elapsedTime.partReq[#j];
                           // add elapsed time
                           #elapsedTime := #elapsedTime + #rt.asReal;
                           // save new value
                           #stations.current[#i].elapsedTime.partReq[#j] := #elapsedTime;
                       END_REGION

                   END_IF;
               END_REGION

           END_FOR;
       END_FOR;
   END_REGION
END_FUNCTION_BLOCK

FUNCTION_BLOCK "Base Animations"   // FB8, SCL
{ S7_Optimized_Access := 'TRUE' }
VERSION : 0.1
   VAR_IN_OUT
      stations : "Stations";
   END_VAR
   VAR_TEMP
      animation : Int;
      i : Int;
      j : Int;
      partRequested : Bool;
      partOrdered : Bool;
      elapsedTime : Real;
      criticalTime : Real;
      alottedTime : Real;
      remainingTime : Real;
   END_VAR
   VAR CONSTANT
      stationCount : Int := 23;
      anDefault : USInt := 0;
      anRequested : USInt := 1;
      anSolidRed : USInt := 2;
      anFlashRed : USInt := 3;
      anPartOrdered : USInt := 4;
   END_VAR
BEGIN
   REGION "MAIN LOOP"
       FOR #i := 0 TO #stationCount DO
           // j := 0 would be the reset button so it is skipped
           FOR #j := 1 TO 7 DO

               REGION "PART REQUEST TIMER"

                   REGION "COPY TO LOCAL"
                       #partRequested := #stations.current[#i].btnStates[#j];
                       #partOrdered := #stations.current[#i].partOrdered[#j];
                   END_REGION

                   REGION "PART REQUESTED"
                       IF #partRequested THEN

                           REGION "GET LOCAL VARIABLES"
                               // remaining time
                               #elapsedTime := #stations.current[#i].elapsedTime.partReq[#j];
                               #alottedTime := #stations.current[#i].presetTime.allotted[#j];
                               #remainingTime := #alottedTime - #elapsedTime;
                               // critical time
                               #criticalTime := #stations.current[#i].presetTime.critical[#j];
                           END_REGION

                           REGION "DEFAULT ANIMATION STATE"
                               IF #remainingTime > #criticalTime THEN
                                   #animation := #anRequested;
                               END_IF;
                           END_REGION

                           REGION "SOLID RED ANIMATION STATE"
                               IF #remainingTime <= #criticalTime AND #elapsedTime > 0.0 THEN
                                   #animation := #anSolidRed;
                               END_IF;
                           END_REGION

                           REGION "FLASHING RED ANIMATION STATE
                               IF #remainingTime <= 0.0 THEN
                                   #animation := #anFlashRed;
                               END_IF;
                           END_REGION ;

                           REGION "ORDERED"
                               IF #partOrdered THEN
                                   #animation := #anPartOrdered;
                               END_IF;
                           END_REGION

                       END_IF;
                   END_REGION

                   REGION "PART NOT REQUESTED"
                       IF NOT #partRequested THEN
                           #animation := #anDefault;
                       END_IF;
                   END_REGION

                   REGION "OUTPUT"
                       #stations.current[#i].animations[#j] := #animation;
                   END_REGION

               END_REGION

           END_FOR;
       END_FOR;
   END_REGION
END_FUNCTION_BLOCK

FUNCTION_BLOCK "Format Part Call Requests"   // FB9, SCL
{ S7_Optimized_Access := 'TRUE' }
VERSION : 0.1
   VAR_INPUT
      constants : "Constants";
   END_VAR
   VAR_IN_OUT
      requests : "Part Request Data";
      stations : "Stations";
   END_VAR
   VAR
      station : Int;
      button : Int;
   END_VAR
   VAR_TEMP
      address : Int;
      animator : UInt;
      maxRows : Int;
      timeAsReal : Real;
      timeAsTime : WString;
      i : Int;
      inStrRslt : Int;
   END_VAR
   VAR CONSTANT
      showSingleLine : UInt := 1;
      showDoubleLine : UInt := 2;
   END_VAR
BEGIN
   // REGION "COPY TO LOCAL"
   //     #maxRows := #constants.partReqRows - 1;
   // END_REGION


   // REGION "ITERATE THROUGH VISIBLE TABLE ROWS"
   //     FOR #i := 0 TO #maxRows DO

   //         REGION "COPY TO LOCAL"
   //             #address := UINT_TO_INT(#requests.row[#i].address);
   //         END_REGION

   //         REGION "HIDE UNPOPULATED ROWS"
   //             IF #address = 0 THEN
   //                 #requests.row[#i].pbSelection.animate := FALSE;
   //                 #requests.row[#i].rtBackground.visibility := FALSE;
   //                 #animator := 0;
   //                 #requests.row[#i].tfDropZone.visibility := FALSE;
   //                 #requests.row[#i].tfDropZone.animate := #animator;
   //                 #requests.row[#i].tfLine.visibility := FALSE;
   //                 #requests.row[#i].tfLine.animate := #animator;
   //                 #requests.row[#i].tfPartNumber.visibility := FALSE;
   //                 #requests.row[#i].tfPartNumber.animate := #animator;
   //                 #requests.row[#i].tfTime.visibility := FALSE;
   //                 #requests.row[#i].tfTime.animate := #animator;
   //             END_IF;
   //         END_REGION

   //         REGION "ANIMATE POPULATED ROWS"

   //             REGION "ANIMATE ROWS WITH DATA"
   //                 IF #address <> 0 THEN

   //                     REGION "GET POINTERS FOR STATION ARRAY"
   //                         #station := #address / 10 - 1;
   //                         #button := #address MOD 10 - 1;
   //                     END_REGION

   //                     REGION "ANIMATIONS"

   //                         REGION "PUSHBUTTON VISIBILITY"
   //                             #requests.row[#i].pbSelection.animate := TRUE;
   //                         END_REGION

   //                         REGION "ANIMATOR VALUE"
   //                             #animator := INT_TO_UINT(#stations.current[#station].animations[#button]);
   //                         END_REGION

   //                         REGION "BACKGROUND VISIBILITY"
   //                             #requests.row[#i].rtBackground.visibility := TRUE;
   //                         END_REGION

   //                         REGION "DROP ZONE" 
   //                             #requests.row[#i].tfDropZone.visibility := TRUE;
   //                             #requests.row[#i].tfDropZone.value := "Strip Sign"(UINT_TO_WSTRING(#stations.current[#station].dropZone));
   //                             #requests.row[#i].tfDropZone.animate := #animator;
   //                         END_REGION

   //                         REGION "LINE"
   //                             #requests.row[#i].tfLine.visibility := TRUE;
   //                             #requests.row[#i].tfLine.value := #stations.current[#station].line;
   //                             #requests.row[#i].tfLine.animate := #animator;
   //                         END_REGION

   //                         REGION "PART NUMBER"
   //                             #requests.row[#i].tfPartNumber.visibility := TRUE;
   //                             #requests.row[#i].tfPartNumber.value := #stations.current[#station].partNumbers[#button];
   //                             #requests.row[#i].tfPartNumber.animate := #animator;
   //                             REGION "DETERMINE VISIBLE ROWS"

   //                                 REGION "FIND CARRIAGE RETURN"
   //                                     #inStrRslt := FIND(IN1 := #requests.row[#i].tfPartNumber.value,
   //                                                        IN2 := wstring#'$L');
   //                                 END_REGION

   //                                 REGION "SINGLE LINE"
   //                                     IF #inStrRslt = 0 THEN
   //                                         #requests.row[#i].tfPartNumber.count := #showSingleLine;
   //                                     END_IF;
   //                                 END_REGION

   //                                 REGION "DOUBLE LINE"
   //                                     IF #inStrRslt <> 0 THEN
   //                                         #requests.row[#i].tfPartNumber.count := #showDoubleLine;
   //                                     END_IF;
   //                                 END_REGION

   //                             END_REGION

   //                         END_REGION

   //                         REGION "TIME"
   //                             #requests.row[#i].tfTime.visibility := TRUE;
   //                             #timeAsReal := #stations.current[#station].presetTime.allotted[#button];
   //                             #timeAsReal -= #stations.current[#station].elapsedTime.partReq[#button];
   //                             #requests.row[#i].tfTime.value := "Real to WString Timer"(#timeAsReal);
   //                             #requests.row[#i].tfTime.animate := #animator;
   //                         END_REGION

   //                     END_REGION

   //                 END_IF;
   //             END_REGION

   //         END_REGION

   //     END_FOR;
   // END_REGION
END_FUNCTION_BLOCK

FUNCTION_BLOCK "KP8 Expanded Animations"   // FB10, SCL
{ S7_Optimized_Access := 'TRUE' }
VERSION : 0.1
   VAR_IN_OUT
      stations : "Stations";
   END_VAR
   VAR_TEMP
      i : Int;
      j : Int;
      colorBox : DWord;
      animation : Int;
      redMask : DWord;
   END_VAR
   VAR CONSTANT
      stationCount : Int := 23;
      buttonCount : Int := 7;
      anSolidRed : USInt := 2;
      anFlashRed : USInt := 3;
   END_VAR
BEGIN
   REGION "LOOP THROUGH STATIONS"
       FOR #i := 0 TO #stationCount DO

           REGION "LOOP THROUGH BUTTONS"
               FOR #j := 0 TO #buttonCount DO

                   REGION "GET ANIMATION"
                       #animation := #stations.current[#i].animations[#j];
                   END_REGION

                   REGION "SOLID RED"
                       IF #animation = #anSolidRed THEN
                           #colorBox := #stations.current[#i].kp8Out;
                           #redMask := 16#FEFEFE00;
                           #redMask := ROL_DWORD(IN := #redMask,
                                                 N := INT_TO_UINT(#j));
                           #colorBox := #colorBox AND #redMask;
                           #redMask := 16#100_0000;
                           #redMask := ROL_DWORD(IN := #redMask,
                                                 N := INT_TO_UINT(#j));
                           #colorBox := #colorBox OR #redMask;
                           #stations.current[#i].kp8Out := #colorBox;
                       END_IF;
                   END_REGION

                   REGION "FLASHING RED"
                       IF #animation = #anFlashRed THEN

                           REGION "RED ON"
                               IF "Clock_1Hz" THEN
                                   #colorBox := #stations.current[#i].kp8Out;
                                   #redMask := 16#FEFEFE00;
                                   #redMask := ROL_DWORD(IN := #redMask,
                                                         N := INT_TO_UINT(#j));
                                   #colorBox := #colorBox AND #redMask;
                                   #redMask := 16#100_0000;
                                   #redMask := ROL_DWORD(IN := #redMask,
                                                         N := INT_TO_UINT(#j));
                                   #colorBox := #colorBox OR #redMask;
                                   #stations.current[#i].kp8Out := #colorBox;
                               END_IF;
                           END_REGION

                           REGION "RED OFF"
                               IF NOT "Clock_1Hz" THEN
                                   #colorBox := #stations.current[#i].kp8Out;
                                   #redMask := 16#FEFEFE00;
                                   #redMask := ROL_DWORD(IN := #redMask,
                                                         N := INT_TO_UINT(#j));
                                   #colorBox := #colorBox AND #redMask;
                                   #stations.current[#i].kp8Out := #colorBox;
                               END_IF;
                           END_REGION

                       END_IF;
                   END_REGION

               END_FOR;
           END_REGION

       END_FOR;
   END_REGION
END_FUNCTION_BLOCK

FUNCTION_BLOCK "Stack Light Animations"   // FB11, SCL
{ S7_Optimized_Access := 'TRUE' }
VERSION : 0.1
   VAR_IN_OUT
      stations : "Stations";
   END_VAR
   VAR_TEMP
      animation : Int;
      i : Int;
      j : Int;
      stackLight : DWord;
   END_VAR
   VAR CONSTANT
      anDefault : USInt := 0;
      anRequested : USInt := 1;
      anSolidRed : USInt := 2;
      anFlashRed : USInt := 3;
      anPartOrdered : USInt := 4;
      buttonCount : Int := 7;
      "Part 01" : Int := 7;
      "Part 01 Green On" : DWord := 16#0400_0000;
      "Part 01 Red On" : DWord := 16#0100_0000;
      "Part 01 Yellow On" : DWord := 16#0200_0000;
      "Part 02" : Int := 3;
      "Part 02 Green On" : DWord := 16#2000_0000;
      "Part 02 Red On" : DWord := 16#0800_0000;
      "Part 02 Yellow On" : DWord := 16#1000_0000;
      "Part 03" : Int := 6;
      "Part 03 Green On" : DWord := 16#0001_0000;
      "Part 03 Red On" : DWord := 16#4000_0000;
      "Part 03 Yellow On" : DWord := 16#8000_0000;
      "Part 04" : Int := 2;
      "Part 04 Green On" : DWord := 16#0008_0000;
      "Part 04 Yellow On" : DWord := 16#0004_0000;
      "Part 04 Red On" : DWord := 16#0002_0000;
      "Part 05" : Int := 5;
      "Part 05 Green On" : DWord := 16#0040_0000;
      "Part 05 Red On" : DWord := 16#0010_0000;
      "Part 05 Yellow On" : DWord := 16#0020_0000;
      "Part 06" : Int := 1;
      "Part 06 Green On" : DWord := 16#0000_0200;
      "Part 06 Red On" : DWord := 16#0080_0000;
      "Part 06 Yellow On" : DWord := 16#0000_0100;
      stationCount : Int := 23;
   END_VAR
BEGIN
   REGION "LOOP THROUGH STATIONS"
       FOR #i := 0 TO #stationCount DO

           REGION "LOOP THROUGH BUTTONS"
               FOR #j := 0 TO #buttonCount DO

                   REGION "COPY INTO LOCAL"
                       #stackLight := #stations.current[#i].stackLightOut;
                       #animation := #stations.current[#i].animations[#j];
                   END_REGION

                   REGION "GREEN"
                       IF #animation = #anDefault THEN
                           CASE #j OF
                               #"Part 01":
                                   #stackLight := #stackLight AND (NOT #"Part 01 Red On");
                                   #stackLight := #stackLight AND (NOT #"Part 01 Yellow On");
                                   #stackLight := #stackLight OR #"Part 01 Green On";
                               #"Part 02":
                                   #stackLight := #stackLight AND (NOT #"Part 02 Red On");
                                   #stackLight := #stackLight AND (NOT #"Part 02 Yellow On");
                                   #stackLight := #stackLight OR #"Part 02 Green On";
                               #"Part 03":
                                   #stackLight := #stackLight AND (NOT #"Part 03 Red On");
                                   #stackLight := #stackLight AND (NOT #"Part 03 Yellow On");
                                   #stackLight := #stackLight OR #"Part 03 Green On";
                               #"Part 04":
                                   #stackLight := #stackLight AND (NOT #"Part 04 Red On");
                                   #stackLight := #stackLight AND (NOT #"Part 04 Yellow On");
                                   #stackLight := #stackLight OR #"Part 04 Green On";
                               #"Part 05":
                                   #stackLight := #stackLight AND (NOT #"Part 05 Red On");
                                   #stackLight := #stackLight AND (NOT #"Part 05 Yellow On");
                                   #stackLight := #stackLight OR #"Part 05 Green On";
                               #"Part 06":
                                   #stackLight := #stackLight AND (NOT #"Part 06 Red On");
                                   #stackLight := #stackLight AND (NOT #"Part 06 Yellow On");
                                   #stackLight := #stackLight OR #"Part 06 Green On";
                               ELSE
                                   ;
                           END_CASE;
                       END_IF;
                   END_REGION

                   REGION "YELLOW"
                       IF #animation = #anRequested THEN
                           CASE #j OF
                               #"Part 01":
                                   #stackLight := #stackLight AND (NOT #"Part 01 Red On");
                                   #stackLight := #stackLight OR #"Part 01 Yellow On";
                                   #stackLight := #stackLight AND (NOT #"Part 01 Green On");
                               #"Part 02":
                                   #stackLight := #stackLight AND (NOT #"Part 02 Red On");
                                   #stackLight := #stackLight OR #"Part 02 Yellow On";
                                   #stackLight := #stackLight AND (NOT #"Part 02 Green On");
                               #"Part 03":
                                   #stackLight := #stackLight AND (NOT #"Part 03 Red On");
                                   #stackLight := #stackLight OR #"Part 03 Yellow On";
                                   #stackLight := #stackLight AND (NOT #"Part 03 Green On");
                               #"Part 04":
                                   #stackLight := #stackLight AND (NOT #"Part 04 Red On");
                                   #stackLight := #stackLight OR #"Part 04 Yellow On";
                                   #stackLight := #stackLight AND (NOT #"Part 04 Green On");
                               #"Part 05":
                                   #stackLight := #stackLight AND (NOT #"Part 05 Red On");
                                   #stackLight := #stackLight OR #"Part 05 Yellow On";
                                   #stackLight := #stackLight AND (NOT #"Part 05 Green On");
                               #"Part 06":
                                   #stackLight := #stackLight AND (NOT #"Part 06 Red On");
                                   #stackLight := #stackLight OR #"Part 06 Yellow On";
                                   #stackLight := #stackLight AND (NOT #"Part 06 Green On");
                               ELSE
                                   ;
                           END_CASE;
                       END_IF;
                   END_REGION

